KUKA KRL program: MyProgram_257().src

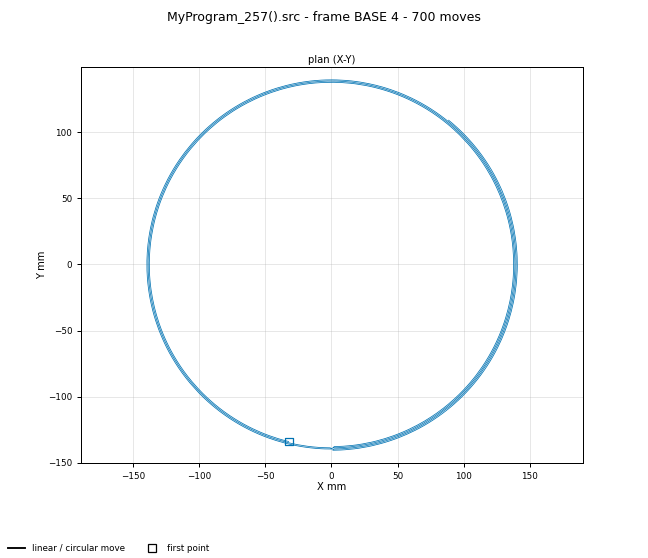
[picture p0: tool path of MyProgram_257().src in frame BASE 4, 700 of 700 moves have a stored position in this frame; points joined in program order, loops and branches not executed]
&ACCESS RVP
&REL 1
&PARAM TEMPLATE = C:\KRC\Roboter\Template\vorgabe
&PARAM EDITMASK = *
DEF MyProgram_257()
; ---- Setting reference (Base) ----
$BASE = BASE_DATA[4]

; --------------------------
; ---- Setting tool (TCP) ----
$TOOL = TOOL_DATA[3]
; --------------------------

$VEL.CP = VEL_APROX_PRINT
Startdeposition()
$VEL.CP = VEL_PRINT
LIN {X -32.383,Y -133.8206,Z 166,A -102.2545,B 10.9184,C 0.327,E1 10.8855,E2 193.1544} C_DIS
LIN {X -35.9329,Y -132.9121,Z 166,A -104.3263,B 10.918,C 0.3387,E1 10.8798,E2 195.2953} C_DIS
LIN {X -40.4402,Y -131.61,Z 166,A -105.7726,B 10.9184,C 0.3257,E1 10.8761,E2 196.6784} C_DIS
LIN {X -44.0124,Y -130.4598,Z 166,A -107.2856,B 10.9185,C 0.3233,E1 10.8721,E2 198.1855} C_DIS
LIN {X -46.9393,Y -129.4346,Z 166,A -108.6006,B 10.9185,C 0.3227,E1 10.8686,E2 199.5036} C_DIS
LIN {X -50.3251,Y -128.1568,Z 166,A -110.1029,B 10.9185,C 0.3213,E1 10.8647,E2 201.0056} C_DIS
LIN {X -53.6285,Y -126.8105,Z 166,A -111.9339,B 10.9184,C 0.3276,E1 10.8598,E2 202.8802} C_DIS
LIN {X -56.9441,Y -125.3576,Z 166,A -113.1055,B 10.9186,C 0.3184,E1 10.857,E2 204.0099} C_DIS
LIN {X -59.558,Y -124.1347,Z 166,A -114.3183,B 10.9186,C 0.3173,E1 10.8539,E2 205.224} C_DIS
LIN {X -62.6311,Y -122.6128,Z 166,A -115.7481,B 10.9187,C 0.3156,E1 10.8503,E2 206.6542} C_DIS
LIN {X -65.7533,Y -120.9695,Z 166,A -117.2938,B 10.9187,C 0.3156,E1 10.8465,E2 208.2095} C_DIS
LIN {X -69.4836,Y -118.8663,Z 166,A -119.1473,B 10.9187,C 0.3147,E1 10.842,E2 210.0718} C_DIS
LIN {X -73.2756,Y -116.5668,Z 166,A -120.9972,B 10.9188,C 0.3122,E1 10.8376,E2 211.9221} C_DIS
LIN {X -77.0533,Y -114.1047,Z 166,A -122.8787,B 10.9189,C 0.3094,E1 10.8332,E2 213.8038} C_DIS
LIN {X -80.9,Y -111.4104,Z 166,A -124.8127,B 10.9189,C 0.3058,E1 10.8288,E2 215.7349} C_DIS
LIN {X -84.5534,Y -108.664,Z 166,A -126.7546,B 10.9191,C 0.3035,E1 10.8245,E2 217.6813} C_DIS
LIN {X -88.1376,Y -105.7781,Z 166,A -128.6782,B 10.9191,C 0.3003,E1 10.8203,E2 219.6055} C_DIS
LIN {X -91.6528,Y -102.7468,Z 166,A -130.3884,B 10.9194,C 0.2919,E1 10.8168,E2 221.2872} C_DIS
LIN {X -94.115,Y -100.4967,Z 166,A -132.0624,B 10.9193,C 0.2955,E1 10.8133,E2 222.9967} C_DIS
LIN {X -97.3746,Y -97.3418,Z 166,A -133.9734,B 10.9193,C 0.2923,E1 10.8095,E2 224.9099} C_DIS
LIN {X -100.6115,Y -93.9917,Z 166,A -135.908,B 10.9195,C 0.2882,E1 10.8058,E2 226.8431} C_DIS
LIN {X -105.5163,Y -88.4499,Z 166,A -138.6237,B 10.9198,C 0.2739,E1 10.8009,E2 229.5118} C_DIS
LIN {X -108.6493,Y -84.5723,Z 166,A -141.1162,B 10.9198,C 0.2782,E1 10.7964,E2 232.0556} C_DIS
LIN {X -111.704,Y -80.4949,Z 166,A -143.216,B 10.9198,C 0.2729,E1 10.7929,E2 234.1518} C_DIS
LIN {X -114.0525,Y -77.1305,Z 166,A -144.9596,B 10.9199,C 0.2696,E1 10.7902,E2 235.8989} C_DIS
LIN {X -116.5303,Y -73.3334,Z 166,A -146.8681,B 10.92,C 0.2655,E1 10.7873,E2 237.8089} C_DIS
LIN {X -118.8585,Y -69.4969,Z 166,A -148.7554,B 10.9201,C 0.2614,E1 10.7846,E2 239.6975} C_DIS
LIN {X -121.0534,Y -65.5995,Z 166,A -150.6918,B 10.9202,C 0.2582,E1 10.782,E2 241.642} C_DIS
LIN {X -122.8275,Y -62.2093,Z 166,A -152.1668,B 10.9204,C 0.2517,E1 10.7801,E2 243.1012} C_DIS
LIN {X -124.3245,Y -59.1608,Z 166,A -153.6073,B 10.9204,C 0.2486,E1 10.7784,E2 244.544} C_DIS
LIN {X -125.811,Y -55.9306,Z 166,A -155.106,B 10.9205,C 0.2451,E1 10.7766,E2 246.044} C_DIS
LIN {X -127.2687,Y -52.5314,Z 166,A -156.6439,B 10.9206,C 0.241,E1 10.775,E2 247.5806} C_DIS
LIN {X -128.6936,Y -48.9386,Z 166,A -158.5186,B 10.9206,C 0.2422,E1 10.773,E2 249.4872} C_DIS
LIN {X -130.2901,Y -44.5133,Z 166,A -160.3071,B 10.9208,C 0.2333,E1 10.7714,E2 251.253} C_DIS
LIN {X -132.3114,Y -38.0805,Z 166,A -163.4175,B 10.9208,C 0.2318,E1 10.7689,E2 254.3987} C_DIS
LIN {X -133.2504,Y -34.6619,Z 166,A -164.5735,B 10.921,C 0.2211,E1 10.7681,E2 255.514} C_DIS
LIN {X -133.8567,Y -32.2332,Z 166,A -165.662,B 10.921,C 0.2191,E1 10.7673,E2 256.6073} C_DIS
LIN {X -134.6523,Y -28.7312,Z 166,A -167.1193,B 10.9212,C 0.2141,E1 10.7664,E2 258.0587} C_DIS
LIN {X -135.2535,Y -25.7509,Z 166,A -168.4646,B 10.9212,C 0.2121,E1 10.7657,E2 259.4127} C_DIS
LIN {X -135.8073,Y -22.6494,Z 166,A -169.7634,B 10.9212,C 0.2081,E1 10.7651,E2 260.7087} C_DIS
LIN {X -136.3093,Y -19.4013,Z 166,A -171.1593,B 10.9213,C 0.2047,E1 10.7645,E2 262.1069} C_DIS
LIN {X -136.7881,Y -15.686,Z 166,A -172.7258,B 10.9214,C 0.2003,E1 10.764,E2 263.6728} C_DIS
LIN {X -137.1684,Y -11.8992,Z 166,A -174.3897,B 10.9214,C 0.1974,E1 10.7636,E2 265.3451} C_DIS
LIN {X -137.432,Y -8.3138,Z 166,A -175.9032,B 10.9215,C 0.1933,E1 10.7633,E2 266.8593} C_DIS
LIN {X -137.6329,Y -3.7244,Z 166,A -177.8392,B 10.9216,C 0.1882,E1 10.7631,E2 268.7963} C_DIS
LIN {X -137.6777,Y 1.4131,Z 166,A -179.9207,B 10.9218,C 0.1808,E1 10.7631,E2 270.8687} C_DIS
LIN {X -137.5612,Y 5.8138,Z 166,A 178.0906,B 10.9218,C 0.1786,E1 10.7632,E2 272.8749} C_DIS
LIN {X -137.262,Y 10.7849,Z 166,A 175.6267,B 10.9218,C 0.1805,E1 10.7637,E2 275.3847} C_DIS
LIN {X -136.9031,Y 14.6358,Z 166,A 174.4183,B 10.922,C 0.1676,E1 10.7641,E2 276.5421} C_DIS
LIN {X -136.4545,Y 18.3583,Z 166,A 172.8363,B 10.922,C 0.1635,E1 10.7646,E2 278.1251} C_DIS
LIN {X -135.8435,Y 22.4325,Z 166,A 171.0426,B 10.922,C 0.1601,E1 10.7654,E2 279.9266} C_DIS
LIN {X -135.2535,Y 25.7509,Z 166,A 169.6825,B 10.9221,C 0.1552,E1 10.7661,E2 281.28} C_DIS
LIN {X -134.5868,Y 29.0346,Z 166,A 168.2737,B 10.9221,C 0.1515,E1 10.7669,E2 282.689} C_DIS
LIN {X -133.7965,Y 32.4827,Z 166,A 166.7901,B 10.9222,C 0.1475,E1 10.7678,E2 284.1724} C_DIS
LIN {X -132.9584,Y 35.7593,Z 166,A 165.3192,B 10.9222,C 0.1448,E1 10.7689,E2 285.6496} C_DIS
LIN {X -132.0104,Y 39.1155,Z 166,A 163.792,B 10.9223,C 0.1422,E1 10.7701,E2 287.1845} C_DIS
LIN {X -130.3953,Y 44.202,Z 166,A 161.4613,B 10.9223,C 0.1382,E1 10.7721,E2 289.5261} C_DIS
LIN {X -129.2183,Y 47.5376,Z 166,A 159.5767,B 10.9223,C 0.1425,E1 10.774,E2 291.4596} C_DIS
LIN {X -127.5636,Y 51.8093,Z 166,A 158.2228,B 10.9225,C 0.126,E1 10.7753,E2 292.7438} C_DIS
LIN {X -126.1563,Y 55.1491,Z 166,A 156.6782,B 10.9225,C 0.1226,E1 10.777,E2 294.2912} C_DIS
LIN {X -124.8829,Y 57.9727,Z 166,A 155.3852,B 10.9225,C 0.1192,E1 10.7785,E2 295.5833} C_DIS
LIN {X -123.0752,Y 61.721,Z 166,A 153.5053,B 10.9226,C 0.1177,E1 10.7808,E2 297.4794} C_DIS
LIN {X -121.5735,Y 64.6289,Z 166,A 152.1846,B 10.9226,C 0.1132,E1 10.7825,E2 298.7936} C_DIS
LIN {X -119.3981,Y 68.5662,Z 166,A 150.2713,B 10.9226,C 0.1092,E1 10.7852,E2 300.7098} C_DIS
LIN {X -117.1399,Y 72.3567,Z 166,A 148.3517,B 10.9227,C 0.1063,E1 10.788,E2 302.6376} C_DIS
LIN {X -114.672,Y 76.2069,Z 166,A 146.4674,B 10.9227,C 0.1012,E1 10.7908,E2 304.5175} C_DIS
LIN {X -112.1852,Y 79.8227,Z 166,A 144.4893,B 10.9227,C 0.0998,E1 10.794,E2 306.512} C_DIS
LIN {X -109.458,Y 83.5227,Z 166,A 142.6774,B 10.9228,C 0.0932,E1 10.797,E2 308.3096} C_DIS
LIN {X -106.6036,Y 87.1364,Z 166,A 140.5684,B 10.9228,C 0.0927,E1 10.8008,E2 310.4399} C_DIS
LIN {X -100.9206,Y 93.6598,Z 166,A 137.4349,B 10.923,C 0.0749,E1 10.8065,E2 313.5126} C_DIS
LIN {X -96.102,Y 98.5982,Z 166,A 133.556,B 10.9229,C 0.0899,E1 10.8143,E2 317.511} C_DIS
LIN {X -91.961,Y 102.4708,Z 166,A 131.8674,B 10.923,C 0.0711,E1 10.8176,E2 319.116} C_DIS
LIN {X -86.1924,Y 107.3687,Z 166,A 128.4073,B 10.923,C 0.0717,E1 10.8251,E2 322.6108} C_DIS
LIN {X -83.4692,Y 109.4985,Z 166,A 127.123,B 10.923,C 0.0658,E1 10.8279,E2 323.8749} C_DIS
LIN {X -80.346,Y 111.811,Z 166,A 124.6738,B 10.923,C 0.0805,E1 10.8338,E2 326.423} C_DIS
LIN {X -74.5833,Y 115.7345,Z 166,A 122.3919,B 10.923,C 0.0626,E1 10.8389,E2 328.6277} C_DIS
LIN {X -71.5622,Y 117.6268,Z 166,A 121.1597,B 10.923,C 0.0549,E1 10.8418,E2 329.828} C_DIS
LIN {X -67.8655,Y 119.7978,Z 166,A 119.3095,B 10.923,C 0.0536,E1 10.8462,E2 331.6847} C_DIS
LIN {X -63.7705,Y 122.0242,Z 166,A 117.1478,B 10.923,C 0.0557,E1 10.8516,E2 333.8715} C_DIS
LIN {X -60.5926,Y 123.6333,Z 166,A 116.0067,B 10.9231,C 0.0463,E1 10.8544,E2 334.9699} C_DIS
LIN {X -57.6179,Y 125.0469,Z 166,A 114.6103,B 10.9231,C 0.045,E1 10.8579,E2 336.3682} C_DIS
LIN {X -54.137,Y 126.5939,Z 166,A 112.7716,B 10.9231,C 0.0487,E1 10.8627,E2 338.2364} C_DIS
LIN {X -49.6794,Y 128.4077,Z 166,A 111.0116,B 10.9231,C 0.0411,E1 10.8672,E2 339.9653} C_DIS
LIN {X -44.9972,Y 130.1223,Z 166,A 108.5657,B 10.9231,C 0.0471,E1 10.8737,E2 342.4547} C_DIS
LIN {X -41.4878,Y 131.2841,Z 166,A 107.5127,B 10.9231,C 0.0349,E1 10.8764,E2 343.4475} C_DIS
LIN {X -38.877,Y 132.0803,Z 166,A 106.2328,B 10.9231,C 0.0371,E1 10.8799,E2 344.7441} C_DIS
LIN {X -35.5788,Y 133.0066,Z 166,A 104.7539,B 10.9231,C 0.0371,E1 10.8838,E2 346.2285} C_DIS
LIN {X -32.1617,Y 133.8739,Z 166,A 103.3043,B 10.9231,C 0.0356,E1 10.8878,E2 347.675} C_DIS
LIN {X -28.2809,Y 134.7495,Z 166,A 101.6915,B 10.9231,C 0.0336,E1 10.8922,E2 349.2816} C_DIS
LIN {X -24.97,Y 135.4018,Z 166,A 100.147,B 10.9231,C 0.0359,E1 10.8964,E2 350.8423} C_DIS
LIN {X -21.0803,Y 136.0597,Z 166,A 98.6216,B 10.9231,C 0.0324,E1 10.9006,E2 352.3523} C_DIS
LIN {X -16.6612,Y 136.6718,Z 166,A 96.2339,B 10.9231,C 0.0437,E1 10.9074,E2 354.8036} C_DIS
LIN {X -12.1006,Y 137.1514,Z 166,A 94.9768,B 10.9231,C 0.0282,E1 10.9107,E2 355.9803} C_DIS
LIN {X -5.5687,Y 137.5707,Z 166,A 92.3656,B 10.9232,C 0.025,E1 10.9179,E2 358.5764} C_DIS
LIN {X 1.7323,Y 137.6735,Z 166,A 89.1943,B 10.9232,C 0.0279,E1 10.9268,E2 361.7628} C_DIS
LIN {X 6.8608,Y 137.5122,Z 166,A 86.8903,B 10.9232,C 0.032,E1 10.9333,E2 364.0865} C_DIS
LIN {X 14.4207,Y 136.9262,Z 166,A 83.7546,B 10.9232,C 0.0322,E1 10.942,E2 367.2187} C_DIS
LIN {X 18.08,Y 136.491,Z 166,A 81.1303,B 10.9231,C 0.0582,E1 10.9497,E2 369.9746} C_DIS
LIN {X 25.8118,Y 135.2419,Z 166,A 79.0317,B 10.9231,C 0.0325,E1 10.955,E2 371.9318} C_DIS
LIN {X 29.0854,Y 134.5758,Z 166,A 77.6421,B 10.9231,C 0.0332,E1 10.9588,E2 373.3209} C_DIS
LIN {X 32.6515,Y 133.7559,Z 166,A 76.026,B 10.9231,C 0.0364,E1 10.9632,E2 374.9482} C_DIS
LIN {X 37.355,Y 132.5189,Z 166,A 74.0809,B 10.9231,C 0.036,E1 10.9684,E2 376.8832} C_DIS
LIN {X 40.4838,Y 131.5966,Z 166,A 72.7493,B 10.9231,C 0.0364,E1 10.972,E2 378.2115} C_DIS
LIN {X 43.8373,Y 130.5181,Z 166,A 71.2639,B 10.9231,C 0.0382,E1 10.9759,E2 379.6991} C_DIS
LIN {X 47.2967,Y 129.3057,Z 166,A 69.7469,B 10.9231,C 0.0394,E1 10.9799,E2 381.2149} C_DIS
LIN {X 51.0221,Y 127.8809,Z 166,A 67.7303,B 10.9231,C 0.0498,E1 10.9853,E2 383.2751} C_DIS
LIN {X 54.4409,Y 126.4625,Z 166,A 66.4824,B 10.9231,C 0.0443,E1 10.9884,E2 384.4872} C_DIS
LIN {X 58.051,Y 124.8467,Z 166,A 64.9058,B 10.9231,C 0.0446,E1 10.9924,E2 386.0553} C_DIS
LIN {X 61.2294,Y 123.3191,Z 166,A 63.4789,B 10.9231,C 0.0454,E1 10.9959,E2 387.4772} C_DIS
LIN {X 64.6818,Y 121.5457,Z 166,A 61.855,B 10.9231,C 0.0477,E1 11,E2 389.1024} C_DIS
LIN {X 68.428,Y 119.477,Z 166,A 60.0037,B 10.9231,C 0.052,E1 11.0045,E2 390.9626} C_DIS
LIN {X 72.3583,Y 117.139,Z 166,A 58.1034,B 10.9231,C 0.0547,E1 11.009,E2 392.8628} C_DIS
LIN {X 76.1504,Y 114.7097,Z 166,A 56.2416,B 10.9231,C 0.0573,E1 11.0134,E2 394.7234} C_DIS
LIN {X 79.8459,Y 112.1686,Z 166,A 54.3732,B 10.9231,C 0.0604,E1 11.0177,E2 396.5923} C_DIS
LIN {X 83.5381,Y 109.4462,Z 166,A 52.4746,B 10.9231,C 0.0634,E1 11.0219,E2 398.4901} C_DIS
LIN {X 87.379,Y 106.4053,Z 166,A 50.2866,B 10.9231,C 0.0709,E1 11.0267,E2 400.6971} C_DIS
LIN {X 89.9112,Y 104.2739,Z 166,A 49.3109,B 10.9231,C 0.0633,E1 11.0287,E2 401.6237} C_DIS
LIN {X 92.6916,Y 101.8106,Z 166,A 47.5978,B 10.9231,C 0.0705,E1 11.0323,E2 403.358} C_DIS
LIN {X 96.7269,Y 97.9856,Z 166,A 45.2698,B 10.923,C 0.0755,E1 11.037,E2 405.6887} C_DIS
LIN {X 102.9757,Y 91.3956,Z 166,A 41.8211,B 10.923,C 0.0749,E1 11.0435,E2 409.0982} C_DIS
LIN {X 105.0773,Y 88.9713,Z 166,A 40.2014,B 10.923,C 0.0852,E1 11.0465,E2 410.7538} C_DIS
LIN {X 107.5009,Y 86.0277,Z 166,A 38.3592,B 10.9228,C 0.0954,E1 11.0498,E2 412.6284} C_DIS
LIN {X 109.8773,Y 82.9702,Z 166,A 37.0695,B 10.9228,C 0.0908,E1 11.0519,E2 413.8792} C_DIS
LIN {X 112.5575,Y 79.2962,Z 166,A 35.2275,B 10.9228,C 0.0939,E1 11.0549,E2 415.716} C_DIS
LIN {X 114.7999,Y 76.0144,Z 166,A 33.5422,B 10.9228,C 0.0987,E1 11.0575,E2 417.4062} C_DIS
LIN {X 117.2171,Y 72.2309,Z 166,A 31.704,B 10.9228,C 0.1025,E1 11.0602,E2 419.2418} C_DIS
LIN {X 120.7526,Y 66.151,Z 166,A 29.0611,B 10.9228,C 0.1024,E1 11.0639,E2 421.8513} C_DIS
LIN {X 122.2935,Y 63.2577,Z 166,A 27.413,B 10.9226,C 0.1134,E1 11.066,E2 423.5358} C_DIS
LIN {X 124.3508,Y 59.1056,Z 166,A 25.6496,B 10.9226,C 0.114,E1 11.0682,E2 425.2799} C_DIS
LIN {X 125.9112,Y 55.7065,Z 166,A 24.1306,B 10.9226,C 0.1172,E1 11.0699,E2 426.7954} C_DIS
LIN {X 127.1624,Y 52.7858,Z 166,A 22.7632,B 10.9226,C 0.1219,E1 11.0714,E2 428.1695} C_DIS
LIN {X 129.6144,Y 46.4406,Z 166,A 20.0434,B 10.9226,C 0.1267,E1 11.0741,E2 430.8776} C_DIS
LIN {X 130.6914,Y 43.3171,Z 166,A 18.6592,B 10.9225,C 0.1307,E1 11.0753,E2 432.2641} C_DIS
LIN {X 131.6878,Y 40.1861,Z 166,A 17.3333,B 10.9225,C 0.1334,E1 11.0764,E2 433.5861} C_DIS
LIN {X 132.6681,Y 36.8215,Z 166,A 15.8877,B 10.9224,C 0.1371,E1 11.0775,E2 435.0313} C_DIS
LIN {X 133.5912,Y 33.3212,Z 166,A 14.4416,B 10.9224,C 0.1398,E1 11.0785,E2 436.4713} C_DIS
LIN {X 134.3803,Y 29.9835,Z 166,A 12.7375,B 10.9222,C 0.1513,E1 11.0796,E2 438.2112} C_DIS
LIN {X 135.2469,Y 25.7854,Z 166,A 11.2256,B 10.9222,C 0.1491,E1 11.0804,E2 439.6907} C_DIS
LIN {X 135.8702,Y 22.2727,Z 166,A 9.7464,B 10.9222,C 0.1532,E1 11.0811,E2 441.1706} C_DIS
LIN {X 136.5716,Y 17.4646,Z 166,A 7.1212,B 10.9218,C 0.1752,E1 11.0821,E2 443.8729} C_DIS
LIN {X 137.142,Y 12.211,Z 166,A 5.6796,B 10.9221,C 0.1614,E1 11.0825,E2 445.2223} C_DIS
LIN {X 137.5808,Y 5.3102,Z 166,A 3.0891,B 10.9221,C 0.1621,E1 11.0829,E2 447.7795} C_DIS
LIN {X 137.6813,Y -0.901,Z 166,A 0.2214,B 10.9218,C 0.1774,E1 11.083,E2 450.6857} C_DIS
LIN {X 137.6128,Y -4.4469,Z 166,A -1.8373,B 10.9215,C 0.1973,E1 11.0828,E2 452.8188} C_DIS
LIN {X 137.3647,Y -9.3811,Z 166,A -3.67,B 10.9215,C 0.1973,E1 11.0825,E2 454.626} C_DIS
LIN {X 137.0563,Y -13.1235,Z 166,A -4.8813,B 10.9215,C 0.1925,E1 11.0822,E2 455.7948} C_DIS
LIN {X 136.6365,Y -16.9568,Z 166,A -7.0897,B 10.9212,C 0.2134,E1 11.0814,E2 458.0806} C_DIS
LIN {X 135.8611,Y -22.3269,Z 166,A -9.3029,B 10.9211,C 0.2188,E1 11.0804,E2 460.2907} C_DIS
LIN {X 134.8829,Y -27.627,Z 166,A -10.8278,B 10.9213,C 0.2061,E1 11.0797,E2 461.728} C_DIS
LIN {X 134.2402,Y -30.5971,Z 166,A -12.1189,B 10.9213,C 0.2105,E1 11.0789,E2 463.0239} C_DIS
LIN {X 133.4197,Y -33.9968,Z 166,A -13.5344,B 10.9212,C 0.2136,E1 11.0779,E2 464.4361} C_DIS
LIN {X 132.4957,Y -37.4382,Z 166,A -14.9407,B 10.9212,C 0.2158,E1 11.0769,E2 465.8343} C_DIS
LIN {X 131.6013,Y -40.4687,Z 166,A -16.2774,B 10.921,C 0.2201,E1 11.0758,E2 467.1752} C_DIS
LIN {X 130.5181,Y -43.8373,Z 166,A -17.7602,B 10.921,C 0.2245,E1 11.0745,E2 468.661} C_DIS
LIN {X 129.2097,Y -47.5607,Z 166,A -19.6751,B 10.9207,C 0.2364,E1 11.0726,E2 470.6121} C_DIS
LIN {X 128.0237,Y -50.6628,Z 166,A -20.7326,B 10.9208,C 0.2316,E1 11.0716,E2 471.6303} C_DIS
LIN {X 126.6556,Y -53.9942,Z 166,A -22.7792,B 10.9204,C 0.2503,E1 11.0693,E2 473.7476} C_DIS
LIN {X 124.6706,Y -58.4317,Z 166,A -24.1138,B 10.9207,C 0.2375,E1 11.0679,E2 474.9979} C_DIS
LIN {X 122.792,Y -62.279,Z 166,A -25.9175,B 10.9206,C 0.2428,E1 11.0656,E2 476.8063} C_DIS
LIN {X 121.0623,Y -65.5831,Z 166,A -27.6131,B 10.9204,C 0.2508,E1 11.0634,E2 478.522} C_DIS
LIN {X 118.8331,Y -69.5401,Z 166,A -29.5854,B 10.9202,C 0.2579,E1 11.0606,E2 480.5068} C_DIS
LIN {X 116.1382,Y -73.9533,Z 166,A -31.6117,B 10.9202,C 0.26,E1 11.0576,E2 482.5196} C_DIS
LIN {X 113.6913,Y -77.6624,Z 166,A -33.4326,B 10.9201,C 0.2639,E1 11.0548,E2 484.339} C_DIS
LIN {X 109.4125,Y -83.5821,Z 166,A -36.1465,B 10.9201,C 0.2627,E1 11.0504,E2 487.015} C_DIS
LIN {X 107.4997,Y -86.0292,Z 166,A -38.1035,B 10.9196,C 0.2833,E1 11.0468,E2 489.0575} C_DIS
LIN {X 104.65,Y -89.474,Z 166,A -39.7777,B 10.9196,C 0.2827,E1 11.0438,E2 490.7103} C_DIS
LIN {X 102.3053,Y -92.1458,Z 166,A -40.7382,B 10.9199,C 0.2724,E1 11.0422,E2 491.6067} C_DIS
LIN {X 99.8387,Y -94.813,Z 166,A -42.5056,B 10.9196,C 0.2825,E1 11.0387,E2 493.4083} C_DIS
LIN {X 96.4271,Y -98.2796,Z 166,A -44.5063,B 10.9196,C 0.2863,E1 11.0348,E2 495.4081} C_DIS
LIN {X 93.2719,Y -101.279,Z 166,A -46.5392,B 10.9193,C 0.2959,E1 11.0306,E2 497.4709} C_DIS
LIN {X 90.6115,Y -103.666,Z 166,A -47.4814,B 10.9196,C 0.2847,E1 11.0287,E2 498.3455} C_DIS
LIN {X 88.2142,Y -105.714,Z 166,A -49.1097,B 10.9193,C 0.2955,E1 11.0252,E2 500.0154} C_DIS
LIN {X 84.6036,Y -108.625,Z 166,A -50.9952,B 10.9193,C 0.2981,E1 11.021,E2 501.8972} C_DIS
LIN {X 79.7823,Y -112.2141,Z 166,A -53.1816,B 10.9193,C 0.2945,E1 11.0162,E2 504.0461} C_DIS
LIN {X 75.6212,Y -115.0588,Z 166,A -56.321,B 10.9185,C 0.3249,E1 11.0086,E2 507.3192} C_DIS
LIN {X 70.1095,Y -118.498,Z 166,A -58.1646,B 10.919,C 0.3074,E1 11.0045,E2 509.0569} C_DIS
LIN {X 64.8573,Y -121.4526,Z 166,A -60.6271,B 10.9189,C 0.3101,E1 10.9985,E2 511.5161} C_DIS
LIN {X 58.3349,Y -124.7154,Z 166,A -63.5408,B 10.9189,C 0.3113,E1 10.9912,E2 514.4171} C_DIS
LIN {X 54.3451,Y -126.5039,Z 166,A -65.484,B 10.9187,C 0.3168,E1 10.9862,E2 516.3776} C_DIS
LIN {X 50.1639,Y -128.2194,Z 166,A -67.4031,B 10.9186,C 0.32,E1 10.9812,E2 518.3031} C_DIS
LIN {X 46.5711,Y -129.5674,Z 166,A -68.8973,B 10.9186,C 0.3193,E1 10.9773,E2 519.7855} C_DIS
LIN {X 43.43,Y -130.6538,Z 166,A -70.276,B 10.9186,C 0.3206,E1 10.9737,E2 521.1647} C_DIS
LIN {X 40.2246,Y -131.676,Z 166,A -71.7112,B 10.9186,C 0.3229,E1 10.9698,E2 522.6055} C_DIS
LIN {X 37.0007,Y -132.618,Z 166,A -73.1007,B 10.9185,C 0.324,E1 10.9661,E2 523.9949} C_DIS
LIN {X 33.7325,Y -133.4868,Z 166,A -74.46,B 10.9185,C 0.324,E1 10.9624,E2 525.3492} C_DIS
LIN {X 30.2325,Y -134.3234,Z 166,A -75.9461,B 10.9185,C 0.3249,E1 10.9584,E2 526.835} C_DIS
LIN {X 23.119,Y -135.729,Z 166,A -78.8202,B 10.9185,C 0.3235,E1 10.9506,E2 529.6929} C_DIS
LIN {X 18.593,Y -136.4237,Z 166,A -81.2342,B 10.9181,C 0.337,E1 10.9437,E2 532.1726} C_DIS
LIN {X 15.0147,Y -136.8623,Z 166,A -83.2047,B 10.9177,C 0.349,E1 10.9381,E2 534.203} C_DIS
LIN {X 8.7523,Y -137.405,Z 166,A -84.7628,B 10.9185,C 0.3243,E1 10.9341,E2 535.629} C_DIS
LIN {X 2.1612,Y -137.6664,Z 166,A -87.7295,B 10.9183,C 0.3304,E1 10.9257,E2 538.6254} C_DIS
LIN {X 2.1612,Y -137.6664,Z 166,A -87.7295,B 10.9183,C 0.3304,E1 10.9257,E2 538.6254} C_DIS
Enddeposition()
LIN {X 0.9873,Y -138.5852,Z 166,A -87.874,B 10.7204,C 0.3366,E1 10.7276,E2 538.8193} C_DIS
Startdeposition()
$VEL.CP = VEL_PRINT
LIN {X 4.4053,Y -138.5308,Z 166,A -85.9781,B 10.7208,C 0.3247,E1 10.733,E2 536.8609} C_DIS
LIN {X 9.1963,Y -138.2958,Z 166,A -83.6201,B 10.7211,C 0.315,E1 10.7398,E2 534.4531} C_DIS
LIN {X 13.343,Y -137.9558,Z 166,A -82.3284,B 10.7208,C 0.3248,E1 10.7432,E2 533.216} C_DIS
LIN {X 20.9166,Y -137.0124,Z 166,A -79.1676,B 10.7208,C 0.323,E1 10.752,E2 530.0527} C_DIS
LIN {X 28.3712,Y -135.6663,Z 166,A -76.0054,B 10.7209,C 0.3202,E1 10.7607,E2 526.8846} C_DIS
LIN {X 32.249,Y -134.7955,Z 166,A -74.468,B 10.7209,C 0.3215,E1 10.7648,E2 525.3598} C_DIS
LIN {X 35.5861,Y -133.953,Z 166,A -73.0543,B 10.7209,C 0.3205,E1 10.7686,E2 523.9462} C_DIS
LIN {X 38.9848,Y -133.0036,Z 166,A -71.5894,B 10.7209,C 0.319,E1 10.7726,E2 522.4794} C_DIS
LIN {X 42.319,Y -131.9806,Z 166,A -70.1924,B 10.7209,C 0.3187,E1 10.7763,E2 521.0871} C_DIS
LIN {X 45.0969,Y -131.0577,Z 166,A -68.9346,B 10.721,C 0.3162,E1 10.7796,E2 519.8222} C_DIS
LIN {X 48.208,Y -129.9458,Z 166,A -67.5456,B 10.7211,C 0.3141,E1 10.7833,E2 518.429} C_DIS
LIN {X 51.3618,Y -128.732,Z 166,A -66.1018,B 10.7211,C 0.3112,E1 10.787,E2 516.9781} C_DIS
LIN {X 54.8665,Y -127.2769,Z 166,A -64.6355,B 10.7211,C 0.3118,E1 10.7908,E2 515.5237} C_DIS
LIN {X 58.6068,Y -125.5993,Z 166,A -62.6121,B 10.7215,C 0.3012,E1 10.796,E2 513.4561} C_DIS
LIN {X 61.908,Y -124.0056,Z 166,A -61.4344,B 10.7213,C 0.3077,E1 10.7989,E2 512.321} C_DIS
LIN {X 65.8602,Y -121.9541,Z 166,A -59.561,B 10.7213,C 0.3041,E1 10.8035,E2 510.4418} C_DIS
LIN {X 69.7841,Y -119.7523,Z 166,A -57.8427,B 10.7213,C 0.3049,E1 10.8076,E2 508.7402} C_DIS
LIN {X 75.5877,Y -116.1757,Z 166,A -54.9111,B 10.7216,C 0.2973,E1 10.8146,E2 505.7914} C_DIS
LIN {X 79.2079,Y -113.7382,Z 166,A -53.2721,B 10.7216,C 0.2984,E1 10.8183,E2 504.172} C_DIS
LIN {X 82.233,Y -111.5702,Z 166,A -51.4175,B 10.7218,C 0.2874,E1 10.8226,E2 502.2748} C_DIS
LIN {X 86.5986,Y -108.2177,Z 166,A -49.2999,B 10.7218,C 0.2871,E1 10.8272,E2 500.1755} C_DIS
LIN {X 90.1572,Y -105.2715,Z 166,A -47.5683,B 10.7218,C 0.288,E1 10.8309,E2 498.4651} C_DIS
LIN {X 93.124,Y -102.6556,Z 166,A -45.7107,B 10.7221,C 0.2788,E1 10.8348,E2 496.5768} C_DIS
LIN {X 96.506,Y -99.483,Z 166,A -43.926,B 10.7221,C 0.2783,E1 10.8384,E2 494.8073} C_DIS
LIN {X 99.7631,Y -96.2167,Z 166,A -42.1277,B 10.7221,C 0.277,E1 10.8419,E2 493.021} C_DIS
LIN {X 101.7923,Y -94.0676,Z 166,A -40.7095,B 10.7223,C 0.2691,E1 10.8446,E2 491.5761} C_DIS
LIN {X 105.2251,Y -90.2111,Z 166,A -38.526,B 10.7225,C 0.2629,E1 10.8486,E2 489.384} C_DIS
LIN {X 107.2815,Y -87.755,Z 166,A -37.4036,B 10.7225,C 0.2651,E1 10.8506,E2 488.2863} C_DIS
LIN {X 110.1177,Y -84.1687,Z 166,A -35.7556,B 10.7224,C 0.2671,E1 10.8534,E2 486.6675} C_DIS
LIN {X 112.8404,Y -80.4819,Z 166,A -33.3227,B 10.7228,C 0.2481,E1 10.8575,E2 484.1627} C_DIS
LIN {X 115.1591,Y -77.1277,Z 166,A -31.9741,B 10.7228,C 0.2529,E1 10.8595,E2 482.8561} C_DIS
LIN {X 117.5029,Y -73.5081,Z 166,A -30.323,B 10.7228,C 0.2519,E1 10.862,E2 481.22} C_DIS
LIN {X 119.6212,Y -70.0077,Z 166,A -28.5457,B 10.7228,C 0.2452,E1 10.8645,E2 479.4297} C_DIS
LIN {X 121.8896,Y -65.9801,Z 166,A -26.6299,B 10.723,C 0.2401,E1 10.8671,E2 477.5111} C_DIS
LIN {X 124.8669,Y -60.1512,Z 166,A -24.1685,B 10.723,C 0.2394,E1 10.8702,E2 475.0782} C_DIS
LIN {X 126.385,Y -56.8917,Z 166,A -22.6797,B 10.7231,C 0.2353,E1 10.8719,E2 473.5875} C_DIS
LIN {X 127.6809,Y -53.9223,Z 166,A -21.2347,B 10.7232,C 0.2288,E1 10.8735,E2 472.1273} C_DIS
LIN {X 128.9804,Y -50.7356,Z 166,A -19.6328,B 10.7234,C 0.2201,E1 10.8752,E2 470.5006} C_DIS
LIN {X 130.136,Y -47.6959,Z 166,A -18.4571,B 10.7234,C 0.2209,E1 10.8763,E2 469.3453} C_DIS
LIN {X 131.4109,Y -44.0569,Z 166,A -17.0402,B 10.7234,C 0.2211,E1 10.8776,E2 467.9494} C_DIS
LIN {X 132.409,Y -40.9609,Z 166,A -15.6068,B 10.7235,C 0.2149,E1 10.8788,E2 466.5031} C_DIS
LIN {X 133.5481,Y -37.0774,Z 166,A -13.9638,B 10.7236,C 0.211,E1 10.88,E2 464.8621} C_DIS
LIN {X 134.67,Y -32.77,Z 166,A -12.2045,B 10.7236,C 0.2079,E1 10.8812,E2 463.1112} C_DIS
LIN {X 135.4404,Y -29.4231,Z 166,A -10.9017,B 10.7236,C 0.2069,E1 10.882,E2 461.8218} C_DIS
LIN {X 136.3221,Y -25.0296,Z 166,A -8.7726,B 10.7239,C 0.1941,E1 10.8832,E2 459.6552} C_DIS
LIN {X 137.1874,Y -19.7347,Z 166,A -6.7708,B 10.7239,C 0.1935,E1 10.884,E2 457.6788} C_DIS
LIN {X 137.6682,Y -16.0447,Z 166,A -5.3556,B 10.7239,C 0.1923,E1 10.8845,E2 456.2778} C_DIS
LIN {X 138.2124,Y -10.3565,Z 166,A -2.6424,B 10.7242,C 0.1759,E1 10.8852,E2 453.5169} C_DIS
LIN {X 138.4225,Y -7.0048,Z 166,A -1.5586,B 10.7242,C 0.1801,E1 10.8853,E2 452.4709} C_DIS
LIN {X 138.5567,Y -3.4728,Z 166,A -0.0225,B 10.7242,C 0.1737,E1 10.8854,E2 450.9236} C_DIS
LIN {X 138.6005,Y 0.4843,Z 166,A 1.8761,B 10.7244,C 0.1619,E1 10.8854,E2 448.9896} C_DIS
LIN {X 138.5332,Y 4.3178,Z 166,A 3.0138,B 10.7244,C 0.1693,E1 10.8854,E2 447.9078} C_DIS
LIN {X 138.2039,Y 10.4731,Z 166,A 5.6782,B 10.7244,C 0.1587,E1 10.8849,E2 445.2261} C_DIS
LIN {X 137.3311,Y 18.722,Z 166,A 8.9179,B 10.7246,C 0.1539,E1 10.8839,E2 442.0075} C_DIS
LIN {X 136.5778,Y 23.5996,Z 166,A 11.0623,B 10.7246,C 0.1452,E1 10.8829,E2 439.848} C_DIS
LIN {X 136.0542,Y 26.4433,Z 166,A 12.1402,B 10.7246,C 0.1449,E1 10.8824,E2 438.7839} C_DIS
LIN {X 135.2605,Y 30.2452,Z 166,A 13.8334,B 10.7248,C 0.138,E1 10.8813,E2 437.078} C_DIS
LIN {X 134.3763,Y 33.9529,Z 166,A 15.2173,B 10.7248,C 0.1387,E1 10.8804,E2 435.7172} C_DIS
LIN {X 133.5522,Y 37.063,Z 166,A 16.5845,B 10.7248,C 0.1339,E1 10.8794,E2 434.3442} C_DIS
LIN {X 132.6522,Y 40.1661,Z 166,A 18.0085,B 10.7248,C 0.1278,E1 10.8783,E2 432.9077} C_DIS
LIN {X 131.6104,Y 43.4576,Z 166,A 19.3215,B 10.7249,C 0.1269,E1 10.8772,E2 431.6082} C_DIS
LIN {X 130.2159,Y 47.4743,Z 166,A 21.4706,B 10.7251,C 0.1117,E1 10.8751,E2 429.4076} C_DIS
LIN {X 128.7625,Y 51.2862,Z 166,A 22.6084,B 10.725,C 0.1217,E1 10.874,E2 428.3386} C_DIS
LIN {X 127.1039,Y 55.2667,Z 166,A 24.4933,B 10.725,C 0.1143,E1 10.8719,E2 426.4393} C_DIS
LIN {X 125.5962,Y 58.6137,Z 166,A 26.106,B 10.7251,C 0.1077,E1 10.87,E2 424.8135} C_DIS
LIN {X 123.6836,Y 62.5476,Z 166,A 27.7851,B 10.7251,C 0.1065,E1 10.868,E2 423.1496} C_DIS
LIN {X 121.9209,Y 65.9219,Z 166,A 29.2087,B 10.7251,C 0.1065,E1 10.8661,E2 421.7439} C_DIS
LIN {X 119.9823,Y 69.3867,Z 166,A 31.3438,B 10.7253,C 0.0893,E1 10.8631,E2 419.545} C_DIS
LIN {X 117.915,Y 72.8457,Z 166,A 32.7107,B 10.7253,C 0.093,E1 10.8611,E2 418.2151} C_DIS
LIN {X 115.5199,Y 76.5873,Z 166,A 34.5301,B 10.7253,C 0.089,E1 10.8584,E2 416.3969} C_DIS
LIN {X 112.9629,Y 80.3106,Z 166,A 36.3702,B 10.7253,C 0.0853,E1 10.8554,E2 414.5591} C_DIS
LIN {X 110.3974,Y 83.8024,Z 166,A 38.487,B 10.7254,C 0.0727,E1 10.8518,E2 412.4} C_DIS
LIN {X 107.7425,Y 87.1887,Z 166,A 39.9838,B 10.7254,C 0.076,E1 10.8492,E2 410.9381} C_DIS
LIN {X 104.3897,Y 91.176,Z 166,A 41.7727,B 10.7254,C 0.0808,E1 10.8461,E2 409.1944} C_DIS
LIN {X 98.427,Y 97.5828,Z 166,A 45.4361,B 10.7254,C 0.0721,E1 10.8391,E2 405.524} C_DIS
LIN {X 94.7146,Y 101.1906,Z 166,A 47.7299,B 10.7254,C 0.0639,E1 10.8344,E2 403.2102} C_DIS
LIN {X 91.445,Y 104.1549,Z 166,A 49.3741,B 10.7254,C 0.065,E1 10.831,E2 401.5881} C_DIS
LIN {X 88.2753,Y 106.8538,Z 166,A 51.1635,B 10.7254,C 0.0601,E1 10.8272,E2 399.7895} C_DIS
LIN {X 84.6632,Y 109.7383,Z 166,A 52.9691,B 10.7254,C 0.0594,E1 10.8232,E2 397.9967} C_DIS
LIN {X 81.7345,Y 111.937,Z 166,A 54.6096,B 10.7255,C 0.0536,E1 10.8195,E2 396.3399} C_DIS
LIN {X 78.0336,Y 114.5478,Z 166,A 56.5105,B 10.7255,C 0.0498,E1 10.8151,E2 394.4351} C_DIS
LIN {X 74.3252,Y 116.988,Z 166,A 58.333,B 10.7255,C 0.0473,E1 10.8109,E2 392.6139} C_DIS
LIN {X 70.4944,Y 119.3353,Z 166,A 60.1676,B 10.7255,C 0.0452,E1 10.8065,E2 390.7818} C_DIS
LIN {X 66.4904,Y 121.6113,Z 166,A 62.0092,B 10.7255,C 0.0441,E1 10.802,E2 388.9479} C_DIS
LIN {X 63.2289,Y 123.3368,Z 166,A 63.4685,B 10.7255,C 0.0437,E1 10.7984,E2 387.4968} C_DIS
LIN {X 60.1286,Y 124.8777,Z 166,A 64.9148,B 10.7255,C 0.0416,E1 10.7948,E2 386.0486} C_DIS
LIN {X 56.9417,Y 126.3626,Z 166,A 66.5886,B 10.7255,C 0.0344,E1 10.7904,E2 384.347} C_DIS
LIN {X 53.9543,Y 127.6676,Z 166,A 67.6164,B 10.7255,C 0.0408,E1 10.7879,E2 383.3595} C_DIS
LIN {X 50.6641,Y 129.0082,Z 166,A 69.1946,B 10.7255,C 0.0366,E1 10.7838,E2 381.7676} C_DIS
LIN {X 47.8414,Y 130.0831,Z 166,A 70.4405,B 10.7255,C 0.0355,E1 10.7805,E2 380.5223} C_DIS
LIN {X 44.0569,Y 131.4109,Z 166,A 72.0272,B 10.7255,C 0.0357,E1 10.7763,E2 378.9446} C_DIS
LIN {X 41.1201,Y 132.3603,Z 166,A 73.3741,B 10.7256,C 0.0329,E1 10.7727,E2 377.5891} C_DIS
LIN {X 37.5816,Y 133.4071,Z 166,A 74.6078,B 10.7256,C 0.0388,E1 10.7695,E2 376.392} C_DIS
LIN {X 34.6308,Y 134.2043,Z 166,A 76.1299,B 10.7256,C 0.0317,E1 10.7653,E2 374.8379} C_DIS
LIN {X 31.0522,Y 135.0762,Z 166,A 77.5139,B 10.7256,C 0.034,E1 10.7616,E2 373.4715} C_DIS
LIN {X 27.9315,Y 135.7561,Z 166,A 78.6952,B 10.7256,C 0.0366,E1 10.7584,E2 372.3079} C_DIS
LIN {X 24.762,Y 136.37,Z 166,A 81.5778,B 10.7256,C -0.0012,E1 10.75,E2 369.2302} C_DIS
LIN {X 15.7453,Y 137.7039,Z 166,A 84.6785,B 10.7256,C 0.0137,E1 10.7416,E2 366.2159} C_DIS
LIN {X 10.3786,Y 138.2108,Z 166,A 86.3123,B 10.7256,C 0.0274,E1 10.7373,E2 364.6578} C_DIS
LIN {X 6.036,Y 138.4696,Z 166,A 87.9842,B 10.7256,C 0.0301,E1 10.7327,E2 363.0025} C_DIS
LIN {X 2.49,Y 138.5774,Z 166,A 89.3697,B 10.7256,C 0.032,E1 10.7288,E2 361.6277} C_DIS
LIN {X -2.9993,Y 138.568,Z 166,A 91.8715,B 10.7256,C 0.0268,E1 10.7218,E2 359.098} C_DIS
LIN {X -8.8912,Y 138.3146,Z 166,A 94.297,B 10.7256,C 0.0275,E1 10.715,E2 356.6753} C_DIS
LIN {X -14.9763,Y 137.7881,Z 166,A 96.879,B 10.7256,C 0.027,E1 10.7078,E2 354.0876} C_DIS
LIN {X -21.4958,Y 136.9227,Z 166,A 99.5067,B 10.7256,C 0.0303,E1 10.7006,E2 351.4729} C_DIS
LIN {X -25.8294,Y 136.1715,Z 166,A 101.0882,B 10.7256,C 0.0367,E1 10.6963,E2 349.9221} C_DIS
LIN {X -29.1823,Y 135.4924,Z 166,A 102.7041,B 10.7256,C 0.0331,E1 10.6918,E2 348.282} C_DIS
LIN {X -32.1671,Y 134.8153,Z 166,A 103.8904,B 10.7256,C 0.0358,E1 10.6886,E2 347.1064} C_DIS
LIN {X -35.5675,Y 133.958,Z 166,A 105.4141,B 10.7256,C 0.0352,E1 10.6845,E2 345.5744} C_DIS
LIN {X -38.8864,Y 133.0324,Z 166,A 106.8289,B 10.7256,C 0.0367,E1 10.6807,E2 344.1619} C_DIS
LIN {X -45.4127,Y 130.9482,Z 166,A 109.6612,B 10.7256,C 0.0394,E1 10.6732,E2 341.3318} C_DIS
LIN {X -48.9184,Y 129.6797,Z 166,A 111.277,B 10.7256,C 0.0394,E1 10.6689,E2 339.708} C_DIS
LIN {X -52.0959,Y 128.4361,Z 166,A 112.9753,B 10.7256,C 0.0346,E1 10.6644,E2 337.9748} C_DIS
LIN {X -55.2632,Y 127.1054,Z 166,A 114.1285,B 10.7256,C 0.0422,E1 10.6616,E2 336.8562} C_DIS
LIN {X -59.3596,Y 125.2451,Z 166,A 115.8813,B 10.7256,C 0.0469,E1 10.6572,E2 335.1182} C_DIS
LIN {X -62.0202,Y 123.9509,Z 166,A 117.2898,B 10.7256,C 0.0445,E1 10.6536,E2 333.6878} C_DIS
LIN {X -66.0088,Y 121.874,Z 166,A 119.2539,B 10.7256,C 0.0449,E1 10.6487,E2 331.7123} C_DIS
LIN {X -70.4495,Y 119.3617,Z 166,A 121.1007,B 10.7256,C 0.0537,E1 10.6443,E2 329.9001} C_DIS
LIN {X -76.0275,Y 115.8884,Z 166,A 123.9149,B 10.7256,C 0.056,E1 10.6377,E2 327.0764} C_DIS
LIN {X -79.337,Y 113.6484,Z 166,A 125.6853,B 10.7256,C 0.0563,E1 10.6336,E2 325.2928} C_DIS
LIN {X -82.5961,Y 111.3023,Z 166,A 127.794,B 10.7256,C 0.0496,E1 10.6287,E2 323.1295} C_DIS
LIN {X -86.2298,Y 108.5113,Z 166,A 129.5207,B 10.7256,C 0.0567,E1 10.625,E2 321.4257} C_DIS
LIN {X -89.0146,Y 106.2388,Z 166,A 130.7739,B 10.7255,C 0.0645,E1 10.6223,E2 320.2031} C_DIS
LIN {X -92.5231,Y 103.1976,Z 166,A 132.5551,B 10.7255,C 0.0713,E1 10.6186,E2 318.4411} C_DIS
LIN {X -96.3475,Y 99.6365,Z 166,A 135.3096,B 10.7255,C 0.0631,E1 10.6129,E2 315.6144} C_DIS
LIN {X -99.5366,Y 96.4507,Z 166,A 136.7733,B 10.7254,C 0.0756,E1 10.6102,E2 314.2029} C_DIS
LIN {X -102.2871,Y 93.5294,Z 166,A 139.0119,B 10.7254,C 0.067,E1 10.6058,E2 311.8933} C_DIS
LIN {X -105.7661,Y 89.576,Z 166,A 140.4757,B 10.7254,C 0.0869,E1 10.6033,E2 310.5213} C_DIS
LIN {X -108.8387,Y 85.8165,Z 166,A 142.7052,B 10.7254,C 0.0869,E1 10.5994,E2 308.2663} C_DIS
LIN {X -111.7441,Y 81.997,Z 166,A 144.693,B 10.7253,C 0.0916,E1 10.5961,E2 306.2801} C_DIS
LIN {X -114.4866,Y 78.1232,Z 166,A 146.697,B 10.7253,C 0.0955,E1 10.5929,E2 304.273} C_DIS
LIN {X -117.0079,Y 74.2936,Z 166,A 148.6222,B 10.7252,C 0.0996,E1 10.5899,E2 302.3462} C_DIS
LIN {X -119.3882,Y 70.4044,Z 166,A 150.5013,B 10.7252,C 0.1045,E1 10.5872,E2 300.4698} C_DIS
LIN {X -121.5829,Y 66.5426,Z 166,A 152.3709,B 10.7252,C 0.1086,E1 10.5847,E2 298.5982} C_DIS
LIN {X -123.4386,Y 63.029,Z 166,A 153.9941,B 10.7251,C 0.1133,E1 10.5826,E2 296.9792} C_DIS
LIN {X -125.2532,Y 59.3426,Z 166,A 155.7814,B 10.7251,C 0.116,E1 10.5804,E2 295.1827} C_DIS
LIN {X -127.078,Y 55.3265,Z 166,A 157.519,B 10.725,C 0.1227,E1 10.5785,E2 293.4579} C_DIS
LIN {X -128.2918,Y 52.454,Z 166,A 159.4945,B 10.725,C 0.1121,E1 10.5764,E2 291.3974} C_DIS
LIN {X -130.2414,Y 47.4035,Z 166,A 160.9014,B 10.7248,C 0.1354,E1 10.5751,E2 290.0977} C_DIS
LIN {X -131.837,Y 42.7685,Z 166,A 163.165,B 10.7248,C 0.1363,E1 10.573,E2 287.8067} C_DIS
LIN {X -132.9681,Y 39.1058,Z 166,A 164.7264,B 10.7248,C 0.1412,E1 10.5718,E2 286.2499} C_DIS
LIN {X -134.216,Y 34.5846,Z 166,A 166.7554,B 10.7247,C 0.1449,E1 10.5703,E2 284.2118} C_DIS
LIN {X -135.1928,Y 30.542,Z 166,A 168.4915,B 10.7247,C 0.1495,E1 10.5692,E2 282.4754} C_DIS
LIN {X -136.0109,Y 26.6694,Z 166,A 170.2189,B 10.7246,C 0.1524,E1 10.5682,E2 280.7384} C_DIS
LIN {X -136.6931,Y 22.9088,Z 166,A 171.6257,B 10.7245,C 0.1605,E1 10.5676,E2 279.355} C_DIS
LIN {X -137.1297,Y 20.1385,Z 166,A 172.9583,B 10.7245,C 0.1603,E1 10.567,E2 278.002} C_DIS
LIN {X -137.6357,Y 16.3176,Z 166,A 174.4542,B 10.7244,C 0.1669,E1 10.5665,E2 276.5199} C_DIS
LIN {X -137.9617,Y 13.2818,Z 166,A 175.8682,B 10.7244,C 0.1675,E1 10.5661,E2 275.0882} C_DIS
LIN {X -138.2865,Y 9.3401,Z 166,A 177.7631,B 10.7244,C 0.167,E1 10.5657,E2 273.1622} C_DIS
LIN {X -138.4749,Y 5.9,Z 166,A 178.9133,B 10.7242,C 0.1768,E1 10.5656,E2 272.0481} C_DIS
LIN {X -138.5793,Y 2.3761,Z 166,A -179.0036,B 10.7243,C 0.1683,E1 10.5655,E2 269.8872} C_DIS
LIN {X -138.5709,Y -2.8849,Z 166,A -177.5225,B 10.724,C 0.1889,E1 10.5655,E2 268.4964} C_DIS
LIN {X -138.4879,Y -5.5683,Z 166,A -176.2365,B 10.724,C 0.1885,E1 10.5656,E2 267.1892} C_DIS
LIN {X -138.2516,Y -9.8188,Z 166,A -174.5162,B 10.724,C 0.1945,E1 10.5659,E2 265.4756} C_DIS
LIN {X -137.972,Y -13.1742,Z 166,A -173.1773,B 10.7238,C 0.1996,E1 10.5663,E2 264.1448} C_DIS
LIN {X -137.6844,Y -15.9091,Z 166,A -171.886,B 10.7238,C 0.1997,E1 10.5667,E2 262.8351} C_DIS
LIN {X -137.1812,Y -19.7778,Z 166,A -170.2588,B 10.7238,C 0.2041,E1 10.5673,E2 261.2075} C_DIS
LIN {X -136.4766,Y -24.1662,Z 166,A -168.4496,B 10.7236,C 0.21,E1 10.5681,E2 259.4036} C_DIS
LIN {X -135.8802,Y -27.3215,Z 166,A -167.2278,B 10.7236,C 0.2159,E1 10.5688,E2 258.1963} C_DIS
LIN {X -135.1434,Y -30.7583,Z 166,A -165.7274,B 10.7234,C 0.2191,E1 10.5697,E2 256.6912} C_DIS
LIN {X -134.3377,Y -34.1051,Z 166,A -163.3595,B 10.7237,C 0.2035,E1 10.5714,E2 254.2042} C_DIS
LIN {X -132.6443,Y -40.1921,Z 166,A -161.6546,B 10.7232,C 0.2297,E1 10.5727,E2 252.6174} C_DIS
LIN {X -131.7587,Y -43.0125,Z 166,A -160.2095,B 10.7232,C 0.2284,E1 10.5739,E2 251.1451} C_DIS
LIN {X -130.6035,Y -46.3993,Z 166,A -158.8961,B 10.7231,C 0.2359,E1 10.5751,E2 249.8539} C_DIS
LIN {X -128.9424,Y -50.8333,Z 166,A -156.706,B 10.7231,C 0.2364,E1 10.5773,E2 247.6358} C_DIS
LIN {X -127.3161,Y -54.776,Z 166,A -155.1084,B 10.7229,C 0.2445,E1 10.579,E2 246.0605} C_DIS
LIN {X -126.0035,Y -57.7328,Z 166,A -153.6502,B 10.7229,C 0.2455,E1 10.5807,E2 244.588} C_DIS
LIN {X -124.3693,Y -61.172,Z 166,A -152.1418,B 10.7228,C 0.2509,E1 10.5825,E2 243.0889} C_DIS
LIN {X -122.8325,Y -64.2025,Z 166,A -150.6802,B 10.7227,C 0.2533,E1 10.5844,E2 241.6211} C_DIS
LIN {X -120.7619,Y -68.0209,Z 166,A -148.7662,B 10.7227,C 0.2554,E1 10.587,E2 239.6933} C_DIS
LIN {X -118.4361,Y -71.9949,Z 166,A -146.8491,B 10.7225,C 0.2598,E1 10.5898,E2 237.7756} C_DIS
LIN {X -116.0026,Y -75.854,Z 166,A -144.9514,B 10.7225,C 0.2641,E1 10.5926,E2 235.8776} C_DIS
LIN {X -113.5955,Y -79.4129,Z 166,A -143.1606,B 10.7223,C 0.2679,E1 10.5955,E2 234.086} C_DIS
LIN {X -111.4615,Y -82.3808,Z 166,A -141.5876,B 10.7223,C 0.2701,E1 10.5981,E2 232.5059} C_DIS
LIN {X -108.7622,Y -85.9138,Z 166,A -139.751,B 10.7222,C 0.2742,E1 10.6012,E2 230.6705} C_DIS
LIN {X -106.1894,Y -89.0735,Z 166,A -137.8763,B 10.7222,C 0.2738,E1 10.6046,E2 228.7722} C_DIS
LIN {X -101.3912,Y -94.4992,Z 166,A -135.0307,B 10.722,C 0.2833,E1 10.6099,E2 225.947} C_DIS
LIN {X -98.6796,Y -97.328,Z 166,A -133.353,B 10.7219,C 0.2854,E1 10.6132,E2 224.2625} C_DIS
LIN {X -95.3605,Y -100.5821,Z 166,A -131.4291,B 10.7219,C 0.289,E1 10.617,E2 222.3391} C_DIS
LIN {X -92.3249,Y -103.3751,Z 166,A -129.9543,B 10.7216,C 0.2973,E1 10.62,E2 220.8943} C_DIS
LIN {X -89.7736,Y -105.5981,Z 166,A -128.3448,B 10.7216,C 0.2952,E1 10.6235,E2 219.2583} C_DIS
LIN {X -86.4123,Y -108.366,Z 166,A -126.5149,B 10.7216,C 0.2977,E1 10.6275,E2 217.4251} C_DIS
LIN {X -82.856,Y -111.1088,Z 166,A -124.6406,B 10.7215,C 0.3004,E1 10.6317,E2 215.5489} C_DIS
LIN {X -79.1417,Y -113.7842,Z 166,A -122.7533,B 10.7215,C 0.3036,E1 10.636,E2 213.6626} C_DIS
LIN {X -75.3749,Y -116.3138,Z 166,A -120.8826,B 10.7213,C 0.3065,E1 10.6403,E2 211.7929} C_DIS
LIN {X -71.6506,Y -118.6443,Z 166,A -119.0156,B 10.7213,C 0.308,E1 10.6448,E2 209.9196} C_DIS
LIN {X -67.699,Y -120.9429,Z 166,A -117.1202,B 10.7213,C 0.3104,E1 10.6494,E2 208.0237} C_DIS
LIN {X -63.6464,Y -123.1241,Z 166,A -115.162,B 10.7212,C 0.3115,E1 10.6542,E2 206.0585} C_DIS
LIN {X -59.4654,Y -125.1946,Z 166,A -113.0007,B 10.7212,C 0.3085,E1 10.6597,E2 203.8671} C_DIS
LIN {X -56.1359,Y -126.723,Z 166,A -111.7803,B 10.721,C 0.3168,E1 10.6627,E2 202.6846} C_DIS
LIN {X -52.7524,Y -128.1695,Z 166,A -110.2629,B 10.721,C 0.3185,E1 10.6667,E2 201.1677} C_DIS
LIN {X -49.12,Y -129.6042,Z 166,A -108.5421,B 10.721,C 0.3175,E1 10.6712,E2 199.433} C_DIS
LIN {X -45.2487,Y -131.0051,Z 166,A -106.9596,B 10.7209,C 0.3217,E1 10.6753,E2 197.8657} C_DIS
LIN {X -41.3021,Y -132.3046,Z 166,A -105.0051,B 10.721,C 0.3176,E1 10.6806,E2 195.8804} C_DIS
LIN {X -34.3015,Y -134.2879,Z 166,A -102.2285,B 10.7208,C 0.3249,E1 10.688,E2 193.1331} C_DIS
LIN {X -30.3625,Y -135.2338,Z 166,A -99.9696,B 10.7212,C 0.3121,E1 10.6944,E2 190.7981} C_DIS
LIN {X -25.6029,Y -136.2148,Z 166,A -98.4516,B 10.7208,C 0.3246,E1 10.6983,E2 189.3433} C_DIS
LIN {X -21.1877,Y -136.9704,Z 166,A -96.6452,B 10.7208,C 0.3263,E1 10.7033,E2 187.5422} C_DIS
LIN {X -18.3547,Y -137.3792,Z 166,A -95.0668,B 10.721,C 0.3172,E1 10.7078,E2 185.9122} C_DIS
LIN {X -14.2983,Y -137.8609,Z 166,A -93.5914,B 10.7209,C 0.3226,E1 10.7118,E2 184.464} C_DIS
LIN {X -9.7705,Y -138.2552,Z 166,A -91.896,B 10.7207,C 0.3272,E1 10.7165,E2 182.7916} C_DIS
LIN {X -5.953,Y -138.4728,Z 166,A -90.2988,B 10.7207,C 0.3268,E1 10.7209,E2 181.1916} C_DIS
LIN {X -1.0065,Y -138.5963,Z 166,A -87.9649,B 10.7209,C 0.3196,E1 10.7276,E2 178.8193} C_DIS
LIN {X -1.0065,Y -138.5963,Z 166,A -87.9649,B 10.7209,C 0.3196,E1 10.7276,E2 178.8193} C_DIS
Enddeposition()
LIN {X 0.9921,Y -139.5084,Z 166,A -87.8538,B 10.7203,C 0.3432,E1 10.7276,E2 178.8349} C_DIS
Startdeposition()
$VEL.CP = VEL_PRINT
LIN {X -2.229,Y -139.4983,Z 166,A -89.3648,B 10.7201,C 0.3479,E1 10.7233,E2 180.3711} C_DIS
LIN {X -4.9101,Y -139.4306,Z 166,A -90.4512,B 10.7201,C 0.3476,E1 10.7202,E2 181.456} C_DIS
LIN {X -7.9201,Y -139.2926,Z 166,A -91.8766,B 10.72,C 0.3521,E1 10.7162,E2 182.9061} C_DIS
LIN {X -11.7893,Y -139.017,Z 166,A -93.3258,B 10.72,C 0.3485,E1 10.7122,E2 184.3374} C_DIS
LIN {X -15.7517,Y -138.6255,Z 166,A -95.1152,B 10.72,C 0.3518,E1 10.7072,E2 186.1473} C_DIS
LIN {X -19.9117,Y -138.0878,Z 166,A -96.7328,B 10.72,C 0.3489,E1 10.7028,E2 187.7519} C_DIS
LIN {X -23.2002,Y -137.5736,Z 166,A -98.1541,B 10.72,C 0.3497,E1 10.6988,E2 189.1806} C_DIS
LIN {X -26.8034,Y -136.9183,Z 166,A -99.6175,B 10.7201,C 0.3481,E1 10.6948,E2 190.6393} C_DIS
LIN {X -31.3518,Y -135.9478,Z 166,A -101.2601,B 10.7203,C 0.3409,E1 10.6904,E2 192.2479} C_DIS
LIN {X -34.5723,Y -135.1646,Z 166,A -103.9201,B 10.7194,C 0.37,E1 10.6828,E2 195.074} C_DIS
LIN {X -41.9125,Y -133.0725,Z 166,A -105.8833,B 10.7203,C 0.341,E1 10.6779,E2 196.8886} C_DIS
LIN {X -44.6171,Y -132.1902,Z 166,A -107.1419,B 10.7203,C 0.3421,E1 10.6746,E2 198.1589} C_DIS
LIN {X -47.4346,Y -131.2044,Z 166,A -108.4183,B 10.7203,C 0.3422,E1 10.6712,E2 199.442} C_DIS
LIN {X -51.5382,Y -129.649,Z 166,A -110.1422,B 10.7203,C 0.3388,E1 10.6667,E2 201.156} C_DIS
LIN {X -55.2995,Y -128.0881,Z 166,A -111.9307,B 10.7203,C 0.3397,E1 10.6621,E2 202.9595} C_DIS
LIN {X -58.5816,Y -126.6206,Z 166,A -113.4332,B 10.7204,C 0.3386,E1 10.6583,E2 204.4653} C_DIS
LIN {X -61.9804,Y -124.9924,Z 166,A -114.9536,B 10.7204,C 0.3362,E1 10.6544,E2 205.9821} C_DIS
LIN {X -65.685,Y -123.0885,Z 166,A -116.7356,B 10.7204,C 0.3357,E1 10.65,E2 207.7733} C_DIS
LIN {X -69.4189,Y -121.0217,Z 166,A -118.489,B 10.7206,C 0.3334,E1 10.6457,E2 209.5266} C_DIS
LIN {X -73.0953,Y -118.837,Z 166,A -120.2523,B 10.7206,C 0.331,E1 10.6415,E2 211.2906} C_DIS
LIN {X -76.6167,Y -116.5977,Z 166,A -122.0007,B 10.7206,C 0.3293,E1 10.6374,E2 213.0432} C_DIS
LIN {X -80.4109,Y -114.0141,Z 166,A -123.9064,B 10.7208,C 0.3268,E1 10.633,E2 214.9511} C_DIS
LIN {X -84.1132,Y -111.3109,Z 166,A -125.7471,B 10.7208,C 0.3227,E1 10.6289,E2 216.786} C_DIS
LIN {X -87.4752,Y -108.6887,Z 166,A -127.5731,B 10.7209,C 0.3214,E1 10.6249,E2 218.6211} C_DIS
LIN {X -90.6791,Y -106.0306,Z 166,A -129.4847,B 10.7209,C 0.3227,E1 10.6208,E2 220.5579} C_DIS
LIN {X -93.1628,Y -103.8549,Z 166,A -130.6582,B 10.7211,C 0.3162,E1 10.6184,E2 221.7077} C_DIS
LIN {X -96.6035,Y -100.6627,Z 166,A -132.6202,B 10.7211,C 0.3132,E1 10.6144,E2 223.6735} C_DIS
LIN {X -99.9564,Y -97.3346,Z 166,A -134.4989,B 10.7213,C 0.308,E1 10.6107,E2 225.5436} C_DIS
LIN {X -106.8625,Y -89.697,Z 166,A -138.8182,B 10.7215,C 0.3011,E1 10.6027,E2 229.8726} C_DIS
LIN {X -109.6985,Y -86.2055,Z 166,A -140.6273,B 10.7216,C 0.2962,E1 10.5995,E2 231.6761} C_DIS
LIN {X -112.6994,Y -82.2446,Z 166,A -142.5123,B 10.7219,C 0.2882,E1 10.5964,E2 233.5402} C_DIS
LIN {X -115.5075,Y -78.2507,Z 166,A -144.778,B 10.7219,C 0.289,E1 10.5927,E2 235.8378} C_DIS
LIN {X -118.0384,Y -74.378,Z 166,A -146.7005,B 10.7219,C 0.2849,E1 10.5898,E2 237.762} C_DIS
LIN {X -120.4499,Y -70.4063,Z 166,A -148.6395,B 10.7221,C 0.2809,E1 10.587,E2 239.7037} C_DIS
LIN {X -122.6857,Y -66.4345,Z 166,A -150.5752,B 10.7221,C 0.2775,E1 10.5844,E2 241.6463} C_DIS
LIN {X -124.5489,Y -62.8679,Z 166,A -152.1005,B 10.7223,C 0.2706,E1 10.5825,E2 243.1543} C_DIS
LIN {X -126.037,Y -59.828,Z 166,A -153.5613,B 10.7223,C 0.2685,E1 10.5807,E2 244.6231} C_DIS
LIN {X -127.5213,Y -56.5956,Z 166,A -155.0166,B 10.7225,C 0.2645,E1 10.579,E2 246.0766} C_DIS
LIN {X -129.2261,Y -52.5873,Z 166,A -156.9849,B 10.7225,C 0.2635,E1 10.5769,E2 248.0662} C_DIS
LIN {X -130.7726,Y -48.6133,Z 166,A -158.7088,B 10.7226,C 0.2582,E1 10.5752,E2 249.7852} C_DIS
LIN {X -132.0167,Y -45.1283,Z 166,A -160.0865,B 10.7228,C 0.2511,E1 10.574,E2 251.1438} C_DIS
LIN {X -132.9982,Y -42.1451,Z 166,A -161.4509,B 10.7228,C 0.2491,E1 10.5728,E2 252.5166} C_DIS
LIN {X -134.2222,Y -38.0697,Z 166,A -163.4758,B 10.7228,C 0.2499,E1 10.5712,E2 254.575} C_DIS
LIN {X -135.0691,Y -34.9487,Z 166,A -164.4728,B 10.723,C 0.2394,E1 10.5705,E2 255.5292} C_DIS
LIN {X -136.1993,Y -30.2504,Z 166,A -166.7201,B 10.723,C 0.2391,E1 10.569,E2 257.8079} C_DIS
LIN {X -137.0648,Y -26.0373,Z 166,A -168.3516,B 10.7232,C 0.2313,E1 10.5682,E2 259.4207} C_DIS
LIN {X -137.659,Y -22.6883,Z 166,A -169.8598,B 10.7232,C 0.2296,E1 10.5675,E2 260.9416} C_DIS
LIN {X -138.2586,Y -18.6967,Z 166,A -171.5817,B 10.7233,C 0.2261,E1 10.5668,E2 262.67} C_DIS
LIN {X -138.7965,Y -14.1708,Z 166,A -173.3267,B 10.7235,C 0.2181,E1 10.5662,E2 264.3974} C_DIS
LIN {X -139.1557,Y -10.0215,Z 166,A -175.1112,B 10.7235,C 0.2146,E1 10.5658,E2 266.1894} C_DIS
LIN {X -139.4415,Y -4.6218,Z 166,A -177.2936,B 10.7237,C 0.2074,E1 10.5656,E2 268.3649} C_DIS
LIN {X -139.4886,Y 2.8166,Z 166,A 179.4251,B 10.7237,C 0.203,E1 10.5656,E2 271.6715} C_DIS
LIN {X -139.2199,Y 9.0998,Z 166,A 176.9694,B 10.724,C 0.1929,E1 10.5659,E2 274.1087} C_DIS
LIN {X -138.6929,Y 15.1333,Z 166,A 174.3459,B 10.724,C 0.1884,E1 10.5666,E2 276.7466} C_DIS
LIN {X -138.1437,Y 19.5206,Z 166,A 172.5793,B 10.7242,C 0.1821,E1 10.5672,E2 278.5051} C_DIS
LIN {X -137.6471,Y 22.7595,Z 166,A 171.1453,B 10.7242,C 0.1799,E1 10.5679,E2 279.9488} C_DIS
LIN {X -136.8448,Y 27.1772,Z 166,A 169.3859,B 10.7243,C 0.1729,E1 10.5688,E2 281.6956} C_DIS
LIN {X -136.2121,Y 30.1909,Z 166,A 168.078,B 10.7243,C 0.1701,E1 10.5695,E2 283.0076} C_DIS
LIN {X -135.5159,Y 33.171,Z 166,A 166.8095,B 10.7244,C 0.1668,E1 10.5704,E2 284.2761} C_DIS
LIN {X -134.6261,Y 36.6187,Z 166,A 165.2018,B 10.7244,C 0.1655,E1 10.5715,E2 285.9004} C_DIS
LIN {X -133.5829,Y 40.2565,Z 166,A 163.8036,B 10.7245,C 0.158,E1 10.5726,E2 287.2774} C_DIS
LIN {X -132.7371,Y 42.9624,Z 166,A 162.5876,B 10.7245,C 0.1557,E1 10.5736,E2 288.4986} C_DIS
LIN {X -131.6271,Y 46.252,Z 166,A 161.1032,B 10.7246,C 0.153,E1 10.575,E2 289.9887} C_DIS
LIN {X -130.3271,Y 49.8005,Z 166,A 159.5553,B 10.7246,C 0.1486,E1 10.5765,E2 291.5344} C_DIS
LIN {X -129.0186,Y 53.0973,Z 166,A 158.1087,B 10.7247,C 0.1444,E1 10.578,E2 292.9781} C_DIS
LIN {X -127.4883,Y 56.6694,Z 166,A 156.1446,B 10.7247,C 0.1475,E1 10.5803,E2 294.9861} C_DIS
LIN {X -126.0885,Y 59.72,Z 166,A 154.9982,B 10.7247,C 0.1391,E1 10.5816,E2 296.1022} C_DIS
LIN {X -123.7599,Y 64.4074,Z 166,A 152.8249,B 10.7249,C 0.1339,E1 10.5843,E2 298.2761} C_DIS
LIN {X -121.7847,Y 68.0715,Z 166,A 151.0332,B 10.7249,C 0.1312,E1 10.5867,E2 300.0762} C_DIS
LIN {X -119.5741,Y 71.884,Z 166,A 149.2692,B 10.7249,C 0.1256,E1 10.5892,E2 301.8324} C_DIS
LIN {X -117.3058,Y 75.529,Z 166,A 147.4119,B 10.7249,C 0.1231,E1 10.592,E2 303.6995} C_DIS
LIN {X -114.734,Y 79.3812,Z 166,A 145.5694,B 10.7251,C 0.1172,E1 10.5949,E2 305.5325} C_DIS
LIN {X -110.6317,Y 85.0051,Z 166,A 141.5025,B 10.7248,C 0.1351,E1 10.602,E2 309.7447} C_DIS
LIN {X -105.4436,Y 91.3611,Z 166,A 139.036,B 10.7251,C 0.109,E1 10.6062,E2 312.097} C_DIS
LIN {X -101.832,Y 95.3705,Z 166,A 136.9242,B 10.7252,C 0.1019,E1 10.6102,E2 314.1936} C_DIS
LIN {X -98.5712,Y 98.7368,Z 166,A 134.9158,B 10.7252,C 0.0996,E1 10.6141,E2 316.2103} C_DIS
LIN {X -95.2303,Y 101.9625,Z 166,A 133.1753,B 10.7252,C 0.0922,E1 10.6176,E2 317.9283} C_DIS
LIN {X -92.6293,Y 104.3313,Z 166,A 131.6746,B 10.7253,C 0.0905,E1 10.6208,E2 319.4344} C_DIS
LIN {X -89.7195,Y 106.8435,Z 166,A 130.0809,B 10.7253,C 0.0877,E1 10.6241,E2 321.0284} C_DIS
LIN {X -86.267,Y 109.6501,Z 166,A 128.1965,B 10.7253,C 0.0855,E1 10.6283,E2 322.918} C_DIS
LIN {X -83.7103,Y 111.6149,Z 166,A 126.8565,B 10.7253,C 0.0834,E1 10.6313,E2 324.2587} C_DIS
LIN {X -80.1844,Y 114.1739,Z 166,A 125.0427,B 10.7253,C 0.0808,E1 10.6354,E2 326.0739} C_DIS
LIN {X -76.8148,Y 116.4673,Z 166,A 123.3556,B 10.7254,C 0.0783,E1 10.6393,E2 327.761} C_DIS
LIN {X -73.2435,Y 118.7459,Z 166,A 121.5832,B 10.7254,C 0.0762,E1 10.6435,E2 329.5358} C_DIS
LIN {X -69.1998,Y 121.1467,Z 166,A 119.4327,B 10.7254,C 0.078,E1 10.6487,E2 331.7116} C_DIS
LIN {X -66.1245,Y 122.8523,Z 166,A 118.2605,B 10.7254,C 0.0701,E1 10.6515,E2 332.849} C_DIS
LIN {X -60.8207,Y 125.5627,Z 166,A 115.8863,B 10.7254,C 0.0652,E1 10.6574,E2 335.2122} C_DIS
LIN {X -58.2427,Y 126.7773,Z 166,A 114.6578,B 10.7254,C 0.065,E1 10.6606,E2 336.4469} C_DIS
LIN {X -54.4264,Y 128.4635,Z 166,A 112.9987,B 10.7255,C 0.0617,E1 10.6648,E2 338.0979} C_DIS
LIN {X -51.3067,Y 129.7415,Z 166,A 111.5731,B 10.7255,C 0.061,E1 10.6685,E2 339.5274} C_DIS
LIN {X -47.9021,Y 131.0358,Z 166,A 110.1383,B 10.7255,C 0.0581,E1 10.6722,E2 340.9534} C_DIS
LIN {X -45.4108,Y 131.9188,Z 166,A 108.8723,B 10.7255,C 0.061,E1 10.6756,E2 342.2409} C_DIS
LIN {X -40.8491,Y 133.4016,Z 166,A 107.0465,B 10.7255,C 0.0559,E1 10.6804,E2 344.0474} C_DIS
LIN {X -37.4416,Y 134.3978,Z 166,A 105.5341,B 10.7255,C 0.0559,E1 10.6845,E2 345.5655} C_DIS
LIN {X -34.354,Y 135.22,Z 166,A 104.1424,B 10.7255,C 0.0567,E1 10.6883,E2 346.9662} C_DIS
LIN {X -29.9835,Y 136.2569,Z 166,A 102.4076,B 10.7255,C 0.0529,E1 10.693,E2 348.6862} C_DIS
LIN {X -25.6267,Y 137.1433,Z 166,A 100.5263,B 10.7255,C 0.053,E1 10.6981,E2 350.5731} C_DIS
LIN {X -20.931,Y 137.9375,Z 166,A 98.3571,B 10.7255,C 0.0569,E1 10.7042,E2 352.7675} C_DIS
LIN {X -15.9417,Y 138.6034,Z 166,A 96.0496,B 10.7255,C 0.0615,E1 10.7107,E2 355.1035} C_DIS
LIN {X -11.9326,Y 139.0049,Z 166,A 94.7639,B 10.7255,C 0.0526,E1 10.7141,E2 356.3427} C_DIS
LIN {X -7.7584,Y 139.3022,Z 166,A 93.1461,B 10.7255,C 0.0499,E1 10.7186,E2 357.9472} C_DIS
LIN {X -4.2627,Y 139.4515,Z 166,A 91.4665,B 10.7255,C 0.0552,E1 10.7233,E2 359.6562} C_DIS
LIN {X 0.7442,Y 139.5141,Z 166,A 89.5713,B 10.7255,C 0.0514,E1 10.7286,E2 361.5304} C_DIS
LIN {X 3.9972,Y 139.4589,Z 166,A 88.1634,B 10.7255,C 0.0531,E1 10.7325,E2 362.9466} C_DIS
LIN {X 7.7118,Y 139.3045,Z 166,A 86.7821,B 10.7255,C 0.0499,E1 10.7363,E2 364.3093} C_DIS
LIN {X 10.5175,Y 139.1195,Z 166,A 85.6092,B 10.7255,C 0.0505,E1 10.7396,E2 365.4839} C_DIS
LIN {X 14.879,Y 138.7203,Z 166,A 83.7947,B 10.7255,C 0.0513,E1 10.7447,E2 367.2998} C_DIS
LIN {X 18.2251,Y 138.3204,Z 166,A 82.3937,B 10.7255,C 0.0521,E1 10.7485,E2 368.7024} C_DIS
LIN {X 22.1045,Y 137.7558,Z 166,A 80.8326,B 10.7255,C 0.0516,E1 10.7528,E2 370.257} C_DIS
LIN {X 28.1493,Y 136.647,Z 166,A 78.2668,B 10.7255,C 0.0539,E1 10.7599,E2 372.8273} C_DIS
LIN {X 33.5163,Y 135.4325,Z 166,A 75.9828,B 10.7255,C 0.0559,E1 10.7661,E2 375.114} C_DIS
LIN {X 38.3481,Y 134.1443,Z 166,A 74.0011,B 10.7255,C 0.0556,E1 10.7714,E2 377.0864} C_DIS
LIN {X 41.3108,Y 133.2603,Z 166,A 72.7484,B 10.7255,C 0.0562,E1 10.7748,E2 378.3367} C_DIS
LIN {X 44.8742,Y 132.1046,Z 166,A 71.0277,B 10.7255,C 0.062,E1 10.7794,E2 380.0799} C_DIS
LIN {X 48.3846,Y 130.8583,Z 166,A 69.7716,B 10.7255,C 0.0568,E1 10.7826,E2 381.3018} C_DIS
LIN {X 50.9299,Y 129.8881,Z 166,A 68.5737,B 10.7255,C 0.0599,E1 10.7857,E2 382.5095} C_DIS
LIN {X 54.6097,Y 128.3863,Z 166,A 66.949,B 10.7255,C 0.0615,E1 10.7899,E2 384.1333} C_DIS
LIN {X 58.0306,Y 126.8754,Z 166,A 65.5107,B 10.7255,C 0.0608,E1 10.7936,E2 385.5592} C_DIS
LIN {X 60.3946,Y 125.7663,Z 166,A 64.3183,B 10.7255,C 0.0651,E1 10.7966,E2 386.7667} C_DIS
LIN {X 63.8069,Y 124.0709,Z 166,A 62.7083,B 10.7255,C 0.0682,E1 10.8006,E2 388.3824} C_DIS
LIN {X 67.6461,Y 122.0211,Z 166,A 60.9154,B 10.7255,C 0.0708,E1 10.805,E2 390.1762} C_DIS
LIN {X 71.5311,Y 119.785,Z 166,A 59.1078,B 10.7255,C 0.0726,E1 10.8094,E2 391.9799} C_DIS
LIN {X 75.0763,Y 117.5955,Z 166,A 57.3747,B 10.7255,C 0.0757,E1 10.8135,E2 393.7159} C_DIS
LIN {X 78.9104,Y 115.0577,Z 166,A 55.5347,B 10.7255,C 0.0775,E1 10.8177,E2 395.5503} C_DIS
LIN {X 82.5273,Y 112.4917,Z 166,A 53.7224,B 10.7254,C 0.0804,E1 10.8218,E2 397.3618} C_DIS
LIN {X 85.3806,Y 110.3418,Z 166,A 52.2533,B 10.7254,C 0.083,E1 10.8251,E2 398.8315} C_DIS
LIN {X 88.7459,Y 107.6541,Z 166,A 50.3381,B 10.7254,C 0.0899,E1 10.8293,E2 400.7655} C_DIS
LIN {X 91.7001,Y 105.1486,Z 166,A 48.9187,B 10.7254,C 0.0885,E1 10.8323,E2 402.164} C_DIS
LIN {X 95.1634,Y 102.0249,Z 166,A 47.0397,B 10.7254,C 0.0913,E1 10.8361,E2 404.0392} C_DIS
LIN {X 97.478,Y 99.8161,Z 166,A 45.7034,B 10.7253,C 0.0945,E1 10.8388,E2 405.3788} C_DIS
LIN {X 100.5271,Y 96.745,Z 166,A 43.9686,B 10.7253,C 0.0971,E1 10.8422,E2 407.109} C_DIS
LIN {X 104.4611,Y 92.4825,Z 166,A 41.7228,B 10.7253,C 0.0986,E1 10.8464,E2 409.3387} C_DIS
LIN {X 106.7863,Y 89.7877,Z 166,A 40.1407,B 10.7252,C 0.105,E1 10.8492,E2 410.9366} C_DIS
LIN {X 109.5701,Y 86.3689,Z 166,A 38.3359,B 10.7252,C 0.1089,E1 10.8524,E2 412.7416} C_DIS
LIN {X 111.5067,Y 83.8538,Z 166,A 37.0773,B 10.7252,C 0.1107,E1 10.8545,E2 413.9953} C_DIS
LIN {X 114.1651,Y 80.1969,Z 166,A 35.2305,B 10.7251,C 0.1148,E1 10.8575,E2 415.8419} C_DIS
LIN {X 116.8378,Y 76.2507,Z 166,A 33.2689,B 10.7251,C 0.1196,E1 10.8605,E2 417.8051} C_DIS
LIN {X 122.0337,Y 67.6233,Z 166,A 29.4051,B 10.725,C 0.1229,E1 10.866,E2 421.6373} C_DIS
LIN {X 123.7039,Y 64.5142,Z 166,A 27.8341,B 10.725,C 0.1297,E1 10.8681,E2 423.2246} C_DIS
LIN {X 125.7144,Y 60.5031,Z 166,A 25.8234,B 10.7248,C 0.1389,E1 10.8706,E2 425.2578} C_DIS
LIN {X 129.926,Y 50.8323,Z 166,A 21.6189,B 10.7247,C 0.1472,E1 10.8752,E2 429.4495} C_DIS
LIN {X 131.3589,Y 47.006,Z 166,A 20.17,B 10.7247,C 0.1457,E1 10.8765,E2 430.8707} C_DIS
LIN {X 132.3839,Y 44.0356,Z 166,A 18.7779,B 10.7247,C 0.1519,E1 10.8778,E2 432.2768} C_DIS
LIN {X 133.6794,Y 39.9379,Z 166,A 17.1437,B 10.7247,C 0.1534,E1 10.8791,E2 433.8959} C_DIS
LIN {X 134.4561,Y 37.2334,Z 166,A 15.9715,B 10.7245,C 0.1571,E1 10.88,E2 435.0712} C_DIS
LIN {X 135.3059,Y 34.0154,Z 166,A 14.639,B 10.7245,C 0.16,E1 10.8809,E2 436.4005} C_DIS
LIN {X 136.1408,Y 30.5069,Z 166,A 12.6491,B 10.7242,C 0.1778,E1 10.8822,E2 438.4562} C_DIS
LIN {X 137.0512,Y 26.1083,Z 166,A 11.5661,B 10.7245,C 0.1628,E1 10.8828,E2 439.4443} C_DIS
LIN {X 138.0386,Y 20.2557,Z 166,A 8.6727,B 10.7242,C 0.182,E1 10.8841,E2 442.398} C_DIS
LIN {X 138.7799,Y 14.3252,Z 166,A 6.5649,B 10.7242,C 0.1798,E1 10.8847,E2 444.4641} C_DIS
LIN {X 139.0876,Y 10.9521,Z 166,A 4.9947,B 10.724,C 0.1887,E1 10.8851,E2 446.0585} C_DIS
LIN {X 139.3723,Y 6.3634,Z 166,A 3.3599,B 10.724,C 0.1874,E1 10.8854,E2 447.6629} C_DIS
LIN {X 139.5047,Y 1.8469,Z 166,A 1.5475,B 10.724,C 0.1917,E1 10.8854,E2 449.4716} C_DIS
LIN {X 139.509,Y -1.5845,Z 166,A 0.1044,B 10.724,C 0.1968,E1 10.8854,E2 450.9206} C_DIS
LIN {X 139.4533,Y -4.1962,Z 166,A -0.9606,B 10.7238,C 0.1997,E1 10.8854,E2 451.9856} C_DIS
LIN {X 139.2811,Y -8.1064,Z 166,A -2.4806,B 10.7238,C 0.2021,E1 10.8852,E2 453.4961} C_DIS
LIN {X 139.056,Y -11.3274,Z 166,A -4,B 10.7236,C 0.2112,E1 10.8849,E2 455.0417} C_DIS
LIN {X 138.7418,Y -14.6787,Z 166,A -5.3075,B 10.7236,C 0.2132,E1 10.8845,E2 456.3411} C_DIS
LIN {X 138.2434,Y -18.8132,Z 166,A -7.0729,B 10.7235,C 0.2197,E1 10.8839,E2 458.1153} C_DIS
LIN {X 137.6109,Y -22.9763,Z 166,A -8.6625,B 10.7235,C 0.221,E1 10.8832,E2 459.689} C_DIS
LIN {X 136.5291,Y -28.7229,Z 166,A -10.9715,B 10.7233,C 0.2255,E1 10.882,E2 461.9888} C_DIS
LIN {X 135.8741,Y -31.6743,Z 166,A -12.2644,B 10.7233,C 0.2304,E1 10.8811,E2 463.2897} C_DIS
LIN {X 135.1509,Y -34.6263,Z 166,A -13.5989,B 10.7231,C 0.2363,E1 10.8802,E2 464.6365} C_DIS
LIN {X 133.846,Y -39.369,Z 166,A -15.515,B 10.7231,C 0.2393,E1 10.8788,E2 466.5416} C_DIS
LIN {X 132.6226,Y -43.3186,Z 166,A -17.1366,B 10.723,C 0.242,E1 10.8774,E2 468.1553} C_DIS
LIN {X 131.352,Y -47.0251,Z 166,A -18.8255,B 10.7228,C 0.2487,E1 10.8758,E2 469.8561} C_DIS
LIN {X 129.7562,Y -51.2692,Z 166,A -20.5547,B 10.7228,C 0.2503,E1 10.8741,E2 471.5705} C_DIS
LIN {X 128.3792,Y -54.6261,Z 166,A -22.0185,B 10.7228,C 0.2537,E1 10.8726,E2 473.0326} C_DIS
LIN {X 127.1899,Y -57.3365,Z 166,A -23.2623,B 10.7226,C 0.2578,E1 10.8711,E2 474.2813} C_DIS
LIN {X 125.4252,Y -61.1029,Z 166,A -25.2902,B 10.7223,C 0.2709,E1 10.8686,E2 476.3521} C_DIS
LIN {X 123.7599,Y -64.4074,Z 166,A -26.2997,B 10.7225,C 0.2613,E1 10.8674,E2 477.2978} C_DIS
LIN {X 122.2917,Y -67.1568,Z 166,A -27.8016,B 10.7223,C 0.2706,E1 10.8654,E2 478.8298} C_DIS
LIN {X 119.9798,Y -71.2043,Z 166,A -30.0068,B 10.722,C 0.2833,E1 10.8622,E2 481.0745} C_DIS
LIN {X 117.8369,Y -74.6973,Z 166,A -31.1849,B 10.7222,C 0.2742,E1 10.8606,E2 482.1897} C_DIS
LIN {X 113.0767,Y -81.7241,Z 166,A -34.7004,B 10.722,C 0.2837,E1 10.855,E2 485.7131} C_DIS
LIN {X 110.82,Y -84.7588,Z 166,A -36.2665,B 10.7219,C 0.2878,E1 10.8524,E2 487.2825} C_DIS
LIN {X 108.367,Y -87.8741,Z 166,A -37.8634,B 10.7218,C 0.2908,E1 10.8496,E2 488.8772} C_DIS
LIN {X 105.8,Y -90.9479,Z 166,A -39.3596,B 10.7218,C 0.2907,E1 10.8469,E2 490.3561} C_DIS
LIN {X 104.1524,Y -92.8299,Z 166,A -40.8567,B 10.7214,C 0.3054,E1 10.844,E2 491.9147} C_DIS
LIN {X 101.5572,Y -95.6623,Z 166,A -42.1079,B 10.7215,C 0.3003,E1 10.8417,E2 493.1257} C_DIS
LIN {X 98.4426,Y -98.8646,Z 166,A -44.0138,B 10.7214,C 0.3062,E1 10.838,E2 495.0427} C_DIS
LIN {X 95.601,Y -101.615,Z 166,A -46.0789,B 10.7209,C 0.3211,E1 10.8337,E2 497.1661} C_DIS
LIN {X 91.7895,Y -105.0706,Z 166,A -47.6422,B 10.7212,C 0.3111,E1 10.8305,E2 498.6612} C_DIS
LIN {X 88.4825,Y -107.8705,Z 166,A -49.515,B 10.7211,C 0.317,E1 10.8265,E2 500.5478} C_DIS
LIN {X 80.904,Y -113.6652,Z 166,A -53.2293,B 10.721,C 0.3191,E1 10.8182,E2 504.2398} C_DIS
LIN {X 77.4805,Y -116.0255,Z 166,A -54.9603,B 10.7209,C 0.3227,E1 10.8142,E2 505.9755} C_DIS
LIN {X 73.0339,Y -118.8747,Z 166,A -57.0419,B 10.7209,C 0.324,E1 10.8093,E2 508.0478} C_DIS
LIN {X 70.0558,Y -120.6539,Z 166,A -58.4814,B 10.7208,C 0.3267,E1 10.8058,E2 509.4906} C_DIS
LIN {X 66.4737,Y -122.6643,Z 166,A -60.2898,B 10.7206,C 0.3324,E1 10.8014,E2 511.3163} C_DIS
LIN {X 62.302,Y -124.8337,Z 166,A -62.4416,B 10.7203,C 0.3407,E1 10.7959,E2 513.4981} C_DIS
LIN {X 58.8787,Y -126.4833,Z 166,A -63.4204,B 10.7207,C 0.3281,E1 10.7937,E2 514.4032} C_DIS
LIN {X 55.0911,Y -128.1782,Z 166,A -65.3144,B 10.7205,C 0.3352,E1 10.7888,E2 516.3233} C_DIS
LIN {X 51.1939,Y -129.7854,Z 166,A -66.9563,B 10.7205,C 0.335,E1 10.7845,E2 517.9551} C_DIS
LIN {X 48.5452,Y -130.7981,Z 166,A -68.1404,B 10.7205,C 0.3369,E1 10.7814,E2 519.1426} C_DIS
LIN {X 45.3905,Y -131.9258,Z 166,A -69.61,B 10.7203,C 0.3407,E1 10.7775,E2 520.6254} C_DIS
LIN {X 41.8456,Y -133.0939,Z 166,A -71.0636,B 10.7203,C 0.3403,E1 10.7737,E2 522.07} C_DIS
LIN {X 38.8763,Y -133.9902,Z 166,A -72.3131,B 10.7203,C 0.3409,E1 10.7703,E2 523.3173} C_DIS
LIN {X 35.6892,Y -134.874,Z 166,A -73.7097,B 10.7203,C 0.3431,E1 10.7666,E2 524.7198} C_DIS
LIN {X 31.5379,Y -135.9053,Z 166,A -75.9171,B 10.7199,C 0.3556,E1 10.7604,E2 526.9864} C_DIS
LIN {X 27.266,Y -136.8267,Z 166,A -77.1627,B 10.7203,C 0.3434,E1 10.7572,E2 528.1626} C_DIS
LIN {X 24.5101,Y -137.346,Z 166,A -78.3688,B 10.7202,C 0.3455,E1 10.7538,E2 529.3765} C_DIS
LIN {X 21.2784,Y -137.8837,Z 166,A -79.7211,B 10.7202,C 0.3465,E1 10.7501,E2 530.7306} C_DIS
LIN {X 17.8779,Y -138.366,Z 166,A -81.1571,B 10.7202,C 0.3478,E1 10.7461,E2 532.1707} C_DIS
LIN {X 11.6992,Y -139.0246,Z 166,A -83.7114,B 10.7201,C 0.349,E1 10.739,E2 534.7269} C_DIS
LIN {X 8.5557,Y -139.2534,Z 166,A -85.0357,B 10.7201,C 0.3501,E1 10.7353,E2 536.0556} C_DIS
LIN {X 4.7311,Y -139.4376,Z 166,A -86.5006,B 10.7201,C 0.3479,E1 10.7313,E2 537.5076} C_DIS
LIN {X 1.9115,Y -139.5036,Z 166,A -87.8082,B 10.72,C 0.3517,E1 10.7276,E2 538.835} C_DIS
LIN {X 1.9115,Y -139.5036,Z 166,A -87.8082,B 10.72,C 0.3517,E1 10.7276,E2 538.835} C_DIS
Enddeposition()
LIN {X 0.9985,Y -140.4282,Z 166,A -87.7386,B 10.7202,C 0.3475,E1 10.7279,E2 538.7427} C_DIS
Startdeposition()
$VEL.CP = VEL_PRINT
LIN {X 3.4546,Y -140.3907,Z 166,A -86.352,B 10.7205,C 0.3379,E1 10.7319,E2 537.3052} C_DIS
LIN {X 6.8938,Y -140.2632,Z 166,A -85.0096,B 10.7205,C 0.339,E1 10.7356,E2 535.9702} C_DIS
LIN {X 10.365,Y -140.0495,Z 166,A -83.5739,B 10.7205,C 0.3382,E1 10.7396,E2 534.5315} C_DIS
LIN {X 14.0283,Y -139.7313,Z 166,A -82.1236,B 10.7205,C 0.3388,E1 10.7437,E2 533.087} C_DIS
LIN {X 17.2049,Y -139.3756,Z 166,A -80.6895,B 10.7205,C 0.3349,E1 10.7477,E2 531.6349} C_DIS
LIN {X 20.8541,Y -138.8767,Z 166,A -79.2889,B 10.7205,C 0.3367,E1 10.7515,E2 530.2469} C_DIS
LIN {X 24.2474,Y -138.324,Z 166,A -77.8935,B 10.7205,C 0.336,E1 10.7554,E2 528.8516} C_DIS
LIN {X 27.6255,Y -137.6887,Z 166,A -76.4983,B 10.7205,C 0.3352,E1 10.7592,E2 527.4563} C_DIS
LIN {X 30.9883,Y -136.9708,Z 166,A -75.0954,B 10.7206,C 0.3341,E1 10.763,E2 526.0525} C_DIS
LIN {X 34.3626,Y -136.1633,Z 166,A -73.6895,B 10.7206,C 0.3332,E1 10.7668,E2 524.6468} C_DIS
LIN {X 37.4666,Y -135.3424,Z 166,A -72.3876,B 10.7206,C 0.3323,E1 10.7703,E2 523.345} C_DIS
LIN {X 41.0097,Y -134.3108,Z 166,A -70.89,B 10.7207,C 0.331,E1 10.7743,E2 521.8473} C_DIS
LIN {X 44.2902,Y -133.265,Z 166,A -69.4922,B 10.7207,C 0.3297,E1 10.7781,E2 520.4494} C_DIS
LIN {X 47.5439,Y -132.1391,Z 166,A -68.0951,B 10.7207,C 0.3284,E1 10.7817,E2 519.0522} C_DIS
LIN {X 50.7692,Y -130.9338,Z 166,A -66.6982,B 10.7208,C 0.327,E1 10.7854,E2 517.6552} C_DIS
LIN {X 53.9639,Y -129.6498,Z 166,A -65.3666,B 10.7208,C 0.3271,E1 10.7888,E2 516.332} C_DIS
LIN {X 57.0121,Y -128.3389,Z 166,A -63.9876,B 10.7208,C 0.3247,E1 10.7923,E2 514.9486} C_DIS
LIN {X 60.1733,Y -126.8876,Z 166,A -62.5868,B 10.7209,C 0.3233,E1 10.7959,E2 513.549} C_DIS
LIN {X 63.1529,Y -125.4321,Z 166,A -61.1715,B 10.721,C 0.3197,E1 10.7994,E2 512.1243} C_DIS
LIN {X 66.3153,Y -123.7901,Z 166,A -59.6576,B 10.7211,C 0.316,E1 10.8032,E2 510.6013} C_DIS
LIN {X 70.0756,Y -121.7013,Z 166,A -57.885,B 10.7212,C 0.3128,E1 10.8075,E2 508.8246} C_DIS
LIN {X 73.7708,Y -119.4978,Z 166,A -56.2669,B 10.7212,C 0.3136,E1 10.8113,E2 507.223} C_DIS
LIN {X 76.6903,Y -117.645,Z 166,A -54.8708,B 10.7212,C 0.3116,E1 10.8146,E2 505.8275} C_DIS
LIN {X 80.158,Y -115.31,Z 166,A -53.1777,B 10.7214,C 0.3089,E1 10.8185,E2 504.1344} C_DIS
LIN {X 83.0825,Y -113.221,Z 166,A -51.6071,B 10.7215,C 0.3035,E1 10.8221,E2 502.5486} C_DIS
LIN {X 86.4996,Y -110.6327,Z 166,A -49.8664,B 10.7215,C 0.3004,E1 10.826,E2 500.8073} C_DIS
LIN {X 89.7567,Y -108.0068,Z 166,A -48.2836,B 10.7215,C 0.3004,E1 10.8293,E2 499.2391} C_DIS
LIN {X 92.4887,Y -105.6767,Z 166,A -46.7195,B 10.7217,C 0.2948,E1 10.8327,E2 497.6603} C_DIS
LIN {X 95.7954,Y -102.6885,Z 166,A -44.958,B 10.7218,C 0.2925,E1 10.8363,E2 495.9045} C_DIS
LIN {X 98.7816,Y -99.8196,Z 166,A -43.2687,B 10.7219,C 0.2889,E1 10.8397,E2 494.2135} C_DIS
LIN {X 101.9495,Y -96.5819,Z 166,A -41.438,B 10.722,C 0.2853,E1 10.8432,E2 492.3831} C_DIS
LIN {X 104.8166,Y -93.4626,Z 166,A -39.7143,B 10.722,C 0.2815,E1 10.8464,E2 490.6582} C_DIS
LIN {X 107.5393,Y -90.3161,Z 166,A -38.0668,B 10.7222,C 0.279,E1 10.8494,E2 489.0154} C_DIS
LIN {X 110.1796,Y -87.0765,Z 166,A -36.4726,B 10.7222,C 0.2779,E1 10.8522,E2 487.434} C_DIS
LIN {X 112.7214,Y -83.7591,Z 166,A -34.7471,B 10.7223,C 0.2733,E1 10.8551,E2 485.7038} C_DIS
LIN {X 115.3248,Y -80.1367,Z 166,A -32.8617,B 10.7225,C 0.267,E1 10.8581,E2 483.8079} C_DIS
LIN {X 117.7186,Y -76.577,Z 166,A -31.1848,B 10.7225,C 0.2646,E1 10.8607,E2 482.1386} C_DIS
LIN {X 120.0023,Y -72.9469,Z 166,A -29.5318,B 10.7225,C 0.2628,E1 10.8631,E2 480.4963} C_DIS
LIN {X 121.7645,Y -69.9663,Z 166,A -28.1089,B 10.7227,C 0.2588,E1 10.8651,E2 479.0706} C_DIS
LIN {X 123.852,Y -66.2001,Z 166,A -26.3782,B 10.7227,C 0.2549,E1 10.8674,E2 477.3413} C_DIS
LIN {X 125.7749,Y -62.4655,Z 166,A -24.6814,B 10.7229,C 0.2508,E1 10.8696,E2 475.6447} C_DIS
LIN {X 127.3202,Y -59.2521,Z 166,A -23.2755,B 10.7229,C 0.2482,E1 10.8712,E2 474.2436} C_DIS
LIN {X 128.4878,Y -56.6792,Z 166,A -22.1387,B 10.7229,C 0.2455,E1 10.8725,E2 473.1077} C_DIS
LIN {X 129.7424,Y -53.7421,Z 166,A -20.846,B 10.723,C 0.2422,E1 10.8739,E2 471.8148} C_DIS
LIN {X 131.0196,Y -50.5484,Z 166,A -19.3622,B 10.7232,C 0.2361,E1 10.8755,E2 470.3188} C_DIS
LIN {X 132.712,Y -45.9205,Z 166,A -17.4428,B 10.7232,C 0.233,E1 10.8772,E2 468.4091} C_DIS
LIN {X 134.0241,Y -41.9452,Z 166,A -15.7964,B 10.7233,C 0.2298,E1 10.8787,E2 466.769} C_DIS
LIN {X 134.9453,Y -38.8755,Z 166,A -14.4447,B 10.7234,C 0.2249,E1 10.8797,E2 465.41} C_DIS
LIN {X 135.8848,Y -35.4554,Z 166,A -13.0422,B 10.7234,C 0.222,E1 10.8807,E2 464.0118} C_DIS
LIN {X 136.8529,Y -31.5046,Z 166,A -11.6586,B 10.7234,C 0.2247,E1 10.8816,E2 462.6623} C_DIS
LIN {X 137.3934,Y -29.0622,Z 166,A -10.4378,B 10.7236,C 0.2163,E1 10.8823,E2 461.4143} C_DIS
LIN {X 138.0646,Y -25.6878,Z 166,A -9.0565,B 10.7236,C 0.2129,E1 10.8831,E2 460.0344} C_DIS
LIN {X 138.653,Y -22.2988,Z 166,A -7.6514,B 10.7237,C 0.2087,E1 10.8837,E2 458.6276} C_DIS
LIN {X 139.1892,Y -18.6483,Z 166,A -6.1535,B 10.7238,C 0.2045,E1 10.8843,E2 457.129} C_DIS
LIN {X 139.5773,Y -15.4802,Z 166,A -4.8849,B 10.7238,C 0.2017,E1 10.8847,E2 455.8634} C_DIS
LIN {X 139.9368,Y -11.7883,Z 166,A -3.403,B 10.7239,C 0.1981,E1 10.8851,E2 454.384} C_DIS
LIN {X 140.1839,Y -8.3552,Z 166,A -2.0536,B 10.7239,C 0.1955,E1 10.8853,E2 453.0402} C_DIS
LIN {X 140.3475,Y -4.9176,Z 166,A -0.6503,B 10.7241,C 0.1914,E1 10.8855,E2 451.6356} C_DIS
LIN {X 140.4271,Y -1.3992,Z 166,A 0.6404,B 10.7241,C 0.1911,E1 10.8855,E2 450.3624} C_DIS
LIN {X 140.4138,Y 2.2956,Z 166,A 2.1412,B 10.7241,C 0.1869,E1 10.8855,E2 448.8609} C_DIS
LIN {X 140.328,Y 5.4168,Z 166,A 3.4858,B 10.7242,C 0.1812,E1 10.8855,E2 447.5057} C_DIS
LIN {X 140.1676,Y 8.6204,Z 166,A 4.8763,B 10.7243,C 0.1751,E1 10.8852,E2 446.1033} C_DIS
LIN {X 139.8938,Y 12.2965,Z 166,A 6.3748,B 10.7244,C 0.1709,E1 10.8848,E2 444.6041} C_DIS
LIN {X 139.5727,Y 15.5228,Z 166,A 7.5969,B 10.7244,C 0.1698,E1 10.8845,E2 443.3938} C_DIS
LIN {X 139.1199,Y 19.1676,Z 166,A 9.098,B 10.7244,C 0.1654,E1 10.8839,E2 441.891} C_DIS
LIN {X 138.608,Y 22.569,Z 166,A 10.4773,B 10.7245,C 0.162,E1 10.8833,E2 440.5135} C_DIS
LIN {X 138.0146,Y 25.9494,Z 166,A 11.8556,B 10.7245,C 0.1586,E1 10.8826,E2 439.1367} C_DIS
LIN {X 137.3395,Y 29.3117,Z 166,A 13.2407,B 10.7246,C 0.1549,E1 10.8819,E2 437.7522} C_DIS
LIN {X 136.5525,Y 32.7817,Z 166,A 14.6468,B 10.7246,C 0.1521,E1 10.881,E2 436.3507} C_DIS
LIN {X 135.7315,Y 36.0302,Z 166,A 16.0638,B 10.7248,C 0.1468,E1 10.88,E2 434.926} C_DIS
LIN {X 134.8735,Y 39.1208,Z 166,A 17.3605,B 10.7248,C 0.1435,E1 10.879,E2 433.6298} C_DIS
LIN {X 133.7985,Y 42.6514,Z 166,A 18.792,B 10.7248,C 0.1413,E1 10.8778,E2 432.2066} C_DIS
LIN {X 132.7124,Y 45.9193,Z 166,A 20.1787,B 10.7248,C 0.138,E1 10.8765,E2 430.8212} C_DIS
LIN {X 131.5295,Y 49.2053,Z 166,A 21.5847,B 10.7249,C 0.1346,E1 10.8752,E2 429.4164} C_DIS
LIN {X 130.2862,Y 52.4087,Z 166,A 22.9678,B 10.7249,C 0.1313,E1 10.8738,E2 428.0347} C_DIS
LIN {X 129.0647,Y 55.3499,Z 166,A 24.2786,B 10.725,C 0.1275,E1 10.8723,E2 426.7214} C_DIS
LIN {X 127.6781,Y 58.4782,Z 166,A 25.6635,B 10.725,C 0.1241,E1 10.8708,E2 425.337} C_DIS
LIN {X 126.2019,Y 61.5998,Z 166,A 27.0169,B 10.725,C 0.1219,E1 10.8691,E2 423.9898} C_DIS
LIN {X 124.5962,Y 64.786,Z 166,A 28.4316,B 10.725,C 0.1193,E1 10.8673,E2 422.5793} C_DIS
LIN {X 122.6501,Y 68.402,Z 166,A 30.1706,B 10.7252,C 0.1133,E1 10.865,E2 420.8311} C_DIS
LIN {X 120.8115,Y 71.5989,Z 166,A 31.7353,B 10.7252,C 0.108,E1 10.8628,E2 419.2576} C_DIS
LIN {X 118.5734,Y 75.2473,Z 166,A 33.4681,B 10.7252,C 0.104,E1 10.8602,E2 417.5255} C_DIS
LIN {X 116.2137,Y 78.8422,Z 166,A 35.1968,B 10.7252,C 0.1005,E1 10.8575,E2 415.7991} C_DIS
LIN {X 113.742,Y 82.3677,Z 166,A 36.9264,B 10.7253,C 0.0971,E1 10.8547,E2 414.072} C_DIS
LIN {X 111.2345,Y 85.7247,Z 166,A 38.5166,B 10.7253,C 0.0963,E1 10.852,E2 412.4963} C_DIS
LIN {X 109.0238,Y 88.5194,Z 166,A 40.0556,B 10.7253,C 0.0908,E1 10.8493,E2 410.9456} C_DIS
LIN {X 106.2566,Y 91.8219,Z 166,A 41.6771,B 10.7253,C 0.0905,E1 10.8464,E2 409.3408} C_DIS
LIN {X 103.9611,Y 94.4128,Z 166,A 43.1972,B 10.7254,C 0.0847,E1 10.8436,E2 407.8062} C_DIS
LIN {X 101.0222,Y 97.5512,Z 166,A 44.9248,B 10.7254,C 0.0817,E1 10.8402,E2 406.0813} C_DIS
LIN {X 97.5497,Y 101.0236,Z 166,A 46.8126,B 10.7254,C 0.0807,E1 10.8365,E2 404.2076} C_DIS
LIN {X 94.4004,Y 103.9724,Z 166,A 48.5569,B 10.7254,C 0.0777,E1 10.8329,E2 402.4648} C_DIS
LIN {X 91.7167,Y 106.3472,Z 166,A 50.0053,B 10.7254,C 0.0753,E1 10.8299,E2 401.0176} C_DIS
LIN {X 88.5186,Y 109.0245,Z 166,A 51.6955,B 10.7255,C 0.0725,E1 10.8262,E2 399.3285} C_DIS
Enddeposition()
END
